LIN {X 0,Y 312.538,Z 248.086,A -85,B 0,C 180,E1 -15604.572,E2 -15604.572} C_VEL
LIN {X 0,Y 312.491,Z 248.051,A -85,B 0,C 180,E1 -15608.073,E2 -15608.073} C_VEL
LIN {X 0,Y 312.47,Z 248.049,A -85,B 0,C 180,E1 -15612.073,E2 -15612.073} C_VEL
LIN {X 0,Y 312.473,Z 248.051,A -85,B 0,C 180,E1 -15616.033,E2 -15616.033} C_VEL
LIN {X 0,Y 312.518,Z 248.056,A -85,B 0,C 180,E1 -15619.872,E2 -15619.872} C_VEL
LIN {X 0,Y 312.546,Z 248.05,A -85,B 0,C 180,E1 -15624.048,E2 -15624.048} C_VEL
LIN {X 0,Y 312.514,Z 248.051,A -85,B 0,C 180,E1 -15627.33,E2 -15627.33} C_VEL
LIN {X 0,Y 312.517,Z 248.049,A -85,B 0,C 180,E1 -15631.289,E2 -15631.289} C_VEL
LIN {X 0,Y 312.528,Z 248.053,A -85,B 0,C 180,E1 -15634.701,E2 -15634.701} C_VEL
LIN {X 0,Y 312.572,Z 248.052,A -85,B 0,C 180,E1 -15637.523,E2 -15637.523} C_VEL
LIN {X 0,Y 312.576,Z 248.049,A -85,B 0,C 180,E1 -15641.647,E2 -15641.647} C_VEL
LIN {X 0,Y 312.693,Z 248.029,A -85,B 0,C 180,E1 -15645.681,E2 -15645.681} C_VEL
LIN {X 0,Y 312.692,Z 248.025,A -85,B 0,C 180,E1 -15649.636,E2 -15649.636} C_VEL
LIN {X 0,Y 312.824,Z 248.015,A -85,B 0,C 180,E1 -15652.248,E2 -15652.248} C_VEL
LIN {X 0,Y 312.702,Z 248.028,A -85,B 0,C 180,E1 -15654.837,E2 -15654.837} C_VEL
LIN {X 0,Y 312.984,Z 247.987,A -85,B 0,C 180,E1 -15658.708,E2 -15658.708} C_VEL
LIN {X 0,Y 312.984,Z 247.997,A -85,B 0,C 180,E1 -15661.281,E2 -15661.281} C_VEL
LIN {X 0,Y 312.701,Z 248.033,A -85,B 0,C 180,E1 -15665.152,E2 -15665.152} C_VEL
LIN {X 0,Y 312.8,Z 248.01,A -85,B 0,C 180,E1 -15667.741,E2 -15667.741} C_VEL
LIN {X 0,Y 312.663,Z 248.028,A -85,B 0,C 180,E1 -15671.665,E2 -15671.665} C_VEL
LIN {X 0,Y 312.659,Z 248.032,A -85,B 0,C 180,E1 -15674.859,E2 -15674.859} C_VEL
LIN {X 0,Y 312.598,Z 248.042,A -85,B 0,C 180,E1 -15679.219,E2 -15679.219} C_VEL
LIN {X 0,Y 312.533,Z 248.052,A -85,B 0,C 180,E1 -15682.783,E2 -15682.783} C_VEL
LIN {X 0,Y 312.581,Z 248.026,A -85,B 0,C 180,E1 -15685.927,E2 -15685.927} C_VEL
LIN {X 0,Y 312.52,Z 248.052,A -85,B 0,C 180,E1 -15689.644,E2 -15689.644} C_VEL
LIN {X 0,Y 312.498,Z 248.057,A -85,B 0,C 180,E1 -15693.683,E2 -15693.683} C_VEL
LIN {X 0,Y 312.531,Z 248.05,A -85,B 0,C 180,E1 -15697.375,E2 -15697.375} C_VEL
LIN {X 0,Y 312.557,Z 248.173,A -85,B 0,C 180,E1 -15699.815,E2 -15699.815} C_VEL
LIN {X 0,Y 314.689,Z 256.545,A -85,B 0,C 180,E1 -15702.93,E2 -15702.93} C_VEL
LIN {X 0,Y 315.577,Z 260.265,A -85,B 0,C 180,E1 -15704.145,E2 -15704.145} C_VEL
LIN {X 0,Y 322.849,Z 275.668,A -85,B 0,C 180,E1 -15705.423,E2 -15705.423} C_VEL
LIN {X 0,Y 325.826,Z 282.967,A -85,B 0,C 180,E1 -15705.933,E2 -15705.933} C_VEL
LIN {X 0,Y 328.456,Z 295.565,A -85,B 0,C 180,E1 -15706.527,E2 -15706.527} C_VEL
LIN {X 0,Y 326.315,Z 367.557,A -85,B 0,C 180,E1 -15708.165,E2 -15708.165} C_VEL
LIN {X 0,Y 325.397,Z 380.734,A -85,B 0,C 180,E1 -15708.693,E2 -15708.693} C_VEL
LIN {X 0,Y 324.242,Z 393.12,A -85,B 0,C 180,E1 -15709.439,E2 -15709.439} C_VEL
LIN {X 0,Y 322.722,Z 405.254,A -85,B 0,C 180,E1 -15710.432,E2 -15710.432} C_VEL
LIN {X 0,Y 321.114,Z 416.236,A -85,B 0,C 180,E1 -15711.609,E2 -15711.609} C_VEL
LIN {X 0,Y 319.402,Z 426.332,A -85,B 0,C 180,E1 -15712.961,E2 -15712.961} C_VEL
LIN {X 0,Y 317.66,Z 435.593,A -85,B 0,C 180,E1 -15714.496,E2 -15714.496} C_VEL
LIN {X 0,Y 316.013,Z 443.977,A -85,B 0,C 180,E1 -15716.221,E2 -15716.221} C_VEL
LIN {X 0,Y 314.401,Z 451.459,A -85,B 0,C 180,E1 -15718.135,E2 -15718.135} C_VEL
LIN {X 0,Y 312.973,Z 458.38,A -85,B 0,C 180,E1 -15720.394,E2 -15720.394} C_VEL
LIN {X 0,Y 311.991,Z 463.287,A -85,B 0,C 180,E1 -15722.497,E2 -15722.497} C_VEL
LIN {X 0,Y 311.343,Z 466.913,A -85,B 0,C 180,E1 -15724.602,E2 -15724.602} C_VEL
LIN {X 0,Y 310.947,Z 468.671,A -85,B 0,C 180,E1 -15725.994,E2 -15725.994} C_VEL
LIN {X 0,Y 310.629,Z 470.416,A -85,B 0,C 180,E1 -15728.046,E2 -15728.046} C_VEL
LIN {X 0,Y 310.434,Z 471.174,A -85,B 0,C 180,E1 -15730.148,E2 -15730.148} C_VEL
LIN {X 0,Y 310.388,Z 471.006,A -85,B 0,C 180,E1 -15731.961,E2 -15731.961} C_VEL
LIN {X 0,Y 310.409,Z 469.679,A -85,B 0,C 180,E1 -15734.235,E2 -15734.235} C_VEL
LIN {X 0,Y 310.678,Z 467.044,A -85,B 0,C 180,E1 -15736.551,E2 -15736.551} C_VEL
LIN {X 0,Y 311.048,Z 462.897,A -85,B 0,C 180,E1 -15738.927,E2 -15738.927} C_VEL
LIN {X 0,Y 311.434,Z 458.154,A -85,B 0,C 180,E1 -15740.911,E2 -15740.911} C_VEL
LIN {X 0,Y 312.152,Z 451.86,A -85,B 0,C 180,E1 -15742.96,E2 -15742.96} C_VEL
LIN {X 0,Y 312.944,Z 444.608,A -85,B 0,C 180,E1 -15744.846,E2 -15744.846} C_VEL
LIN {X 0,Y 313.812,Z 436.952,A -85,B 0,C 180,E1 -15746.469,E2 -15746.469} C_VEL
LIN {X 0,Y 314.939,Z 427.65,A -85,B 0,C 180,E1 -15748.081,E2 -15748.081} C_VEL
LIN {X 0,Y 316.222,Z 416.808,A -85,B 0,C 180,E1 -15749.576,E2 -15749.576} C_VEL
LIN {X 0,Y 317.338,Z 405.733,A -85,B 0,C 180,E1 -15750.793,E2 -15750.793} C_VEL
LIN {X 0,Y 318.354,Z 393.728,A -85,B 0,C 180,E1 -15751.818,E2 -15751.818} C_VEL
LIN {X 0,Y 319.171,Z 381.15,A -85,B 0,C 180,E1 -15752.603,E2 -15752.603} C_VEL
LIN {X 0,Y 319.821,Z 368.153,A -85,B 0,C 180,E1 -15753.149,E2 -15753.149} C_VEL
LIN {X 0,Y 321.21,Z 306.929,A -85,B 0,C 180,E1 -15754.552,E2 -15754.552} C_VEL
LIN {X 0,Y 321.345,Z 291.631,A -85,B 0,C 180,E1 -15754.905,E2 -15754.905} C_VEL
LIN {X 0,Y 317.139,Z 266.964,A -85,B 0,C 180,E1 -15755.749,E2 -15755.749} C_VEL
LIN {X 0,Y 314.935,Z 260.111,A -85,B 0,C 180,E1 -15756.093,E2 -15756.093} C_VEL
LIN {X 0,Y 313.686,Z 252.533,A -85,B 0,C 180,E1 -15758.373,E2 -15758.373} C_VEL
LIN {X 0,Y 312.752,Z 248.06,A -85,B 0,C 180,E1 -15759.906,E2 -15759.906} C_VEL
LIN {X 0,Y 312.663,Z 248.034,A -85,B 0,C 180,E1 -15764.315,E2 -15764.315} C_VEL
LIN {X 0,Y 312.606,Z 248.027,A -85,B 0,C 180,E1 -15768.345,E2 -15768.345} C_VEL
LIN {X 0,Y 312.59,Z 248.047,A -85,B 0,C 180,E1 -15772.47,E2 -15772.47} C_VEL
LIN {X 0,Y 312.564,Z 248.018,A -85,B 0,C 180,E1 -15775.939,E2 -15775.939} C_VEL
LIN {X 0,Y 312.524,Z 248.044,A -85,B 0,C 180,E1 -15779.651,E2 -15779.651} C_VEL
LIN {X 0,Y 312.542,Z 248.048,A -85,B 0,C 180,E1 -15783.709,E2 -15783.709} C_VEL
LIN {X 0,Y 312.554,Z 248.049,A -85,B 0,C 180,E1 -15787.38,E2 -15787.38} C_VEL
LIN {X 0,Y 312.532,Z 248.048,A -85,B 0,C 180,E1 -15789.862,E2 -15789.862} C_VEL
LIN {X 0,Y 311.896,Z 248.126,A -85,B 0,C 180,E1 -15790.938,E2 -15790.938} C_VEL
LIN {X 0,Y 309.08,Z 248.479,A -85,B 0,C 180,E1 -15792.691,E2 -15792.691} C_VEL
LIN {X 0,Y 306.665,Z 248.781,A -85,B 0,C 180,E1 -15794.112,E2 -15794.112} C_VEL
LIN {X 0,Y 305.608,Z 248.913,A -85,B 0,C 180,E1 -15795.212,E2 -15795.212} C_VEL
LIN {X 0,Y 305.512,Z 248.925,A -85,B 0,C 180,E1 -15795.584,E2 -15795.584} C_VEL
LIN {X 0,Y 305.458,Z 248.925,A -85,B 0,C 180,E1 -15799.399,E2 -15799.399} C_VEL
LIN {X 0,Y 305.476,Z 248.918,A -85,B 0,C 180,E1 -15803.27,E2 -15803.27} C_VEL
LIN {X 0,Y 305.442,Z 248.939,A -85,B 0,C 180,E1 -15806.489,E2 -15806.489} C_VEL
LIN {X 0,Y 305.444,Z 248.926,A -85,B 0,C 180,E1 -15809.597,E2 -15809.597} C_VEL
LIN {X 0,Y 305.501,Z 248.895,A -85,B 0,C 180,E1 -15812.615,E2 -15812.615} C_VEL
LIN {X 0,Y 305.493,Z 248.922,A -85,B 0,C 180,E1 -15815.545,E2 -15815.545} C_VEL
LIN {X 0,Y 305.518,Z 248.923,A -85,B 0,C 180,E1 -15819.822,E2 -15819.822} C_VEL
LIN {X 0,Y 305.561,Z 248.899,A -85,B 0,C 180,E1 -15822.609,E2 -15822.609} C_VEL
LIN {X 0,Y 305.637,Z 248.874,A -85,B 0,C 180,E1 -15825.355,E2 -15825.355} C_VEL
LIN {X 0,Y 305.632,Z 248.91,A -85,B 0,C 180,E1 -15829.406,E2 -15829.406} C_VEL
LIN {X 0,Y 305.805,Z 248.889,A -85,B 0,C 180,E1 -15832.08,E2 -15832.08} C_VEL
LIN {X 0,Y 305.683,Z 248.895,A -85,B 0,C 180,E1 -15834.73,E2 -15834.73} C_VEL
LIN {X 0,Y 305.951,Z 248.838,A -85,B 0,C 180,E1 -15838.69,E2 -15838.69} C_VEL
LIN {X 0,Y 305.953,Z 248.861,A -85,B 0,C 180,E1 -15841.322,E2 -15841.322} C_VEL
LIN {X 0,Y 305.674,Z 248.907,A -85,B 0,C 180,E1 -15845.282,E2 -15845.282} C_VEL
LIN {X 0,Y 305.752,Z 248.88,A -85,B 0,C 180,E1 -15847.933,E2 -15847.933} C_VEL
LIN {X 0,Y 305.601,Z 248.893,A -85,B 0,C 180,E1 -15851.951,E2 -15851.951} C_VEL
LIN {X 0,Y 305.642,Z 248.91,A -85,B 0,C 180,E1 -15855.04,E2 -15855.04} C_VEL
LIN {X 0,Y 305.585,Z 248.906,A -85,B 0,C 180,E1 -15858.788,E2 -15858.788} C_VEL
LIN {X 0,Y 305.493,Z 248.921,A -85,B 0,C 180,E1 -15863.044,E2 -15863.044} C_VEL
LIN {X 0,Y 305.531,Z 248.928,A -85,B 0,C 180,E1 -15866.222,E2 -15866.222} C_VEL
LIN {X 0,Y 305.479,Z 248.915,A -85,B 0,C 180,E1 -15869.046,E2 -15869.046} C_VEL
LIN {X 0,Y 305.446,Z 248.933,A -85,B 0,C 180,E1 -15871.957,E2 -15871.957} C_VEL
LIN {X 0,Y 305.471,Z 248.933,A -85,B 0,C 180,E1 -15875.117,E2 -15875.117} C_VEL
LIN {X 0,Y 305.445,Z 248.93,A -85,B 0,C 180,E1 -15878.529,E2 -15878.529} C_VEL
LIN {X 0,Y 305.451,Z 248.928,A -85,B 0,C 180,E1 -15881.861,E2 -15881.861} C_VEL
LIN {X 0,Y 305.411,Z 248.902,A -85,B 0,C 180,E1 -15885.515,E2 -15885.515} C_VEL
LIN {X 0,Y 305.424,Z 248.934,A -85,B 0,C 180,E1 -15888.141,E2 -15888.141} C_VEL
LIN {X 0,Y 305.457,Z 248.925,A -85,B 0,C 180,E1 -15891.595,E2 -15891.595} C_VEL
LIN {X 0,Y 305.475,Z 248.932,A -85,B 0,C 180,E1 -15894.889,E2 -15894.889} C_VEL
LIN {X 0,Y 305.456,Z 248.932,A -85,B 0,C 180,E1 -15898.361,E2 -15898.361} C_VEL
LIN {X 0,Y 305.56,Z 249.121,A -85,B 0,C 180,E1 -15899.775,E2 -15899.775} C_VEL
LIN {X 0,Y 307.636,Z 259.297,A -85,B 0,C 180,E1 -15903.002,E2 -15903.002} C_VEL
LIN {X 0,Y 308.973,Z 267.763,A -85,B 0,C 180,E1 -15905.519,E2 -15905.519} C_VEL
LIN {X 0,Y 309.608,Z 272.24,A -85,B 0,C 180,E1 -15905.741,E2 -15905.741} C_VEL
LIN {X 0,Y 314.56,Z 305.462,A -85,B 0,C 180,E1 -15906.861,E2 -15906.861} C_VEL
LIN {X 0,Y 313.094,Z 375.459,A -85,B 0,C 180,E1 -15908.478,E2 -15908.478} C_VEL
LIN {X 0,Y 312.383,Z 388.794,A -85,B 0,C 180,E1 -15909.032,E2 -15909.032} C_VEL
LIN {X 0,Y 311.352,Z 402.15,A -85,B 0,C 180,E1 -15909.866,E2 -15909.866} C_VEL
LIN {X 0,Y 310.293,Z 413.361,A -85,B 0,C 180,E1 -15910.828,E2 -15910.828} C_VEL
LIN {X 0,Y 308.976,Z 425.009,A -85,B 0,C 180,E1 -15912.118,E2 -15912.118} C_VEL
LIN {X 0,Y 307.955,Z 434.567,A -85,B 0,C 180,E1 -15913.448,E2 -15913.448} C_VEL
LIN {X 0,Y 306.817,Z 444.067,A -85,B 0,C 180,E1 -15915.067,E2 -15915.067} C_VEL
LIN {X 0,Y 305.827,Z 451.94,A -85,B 0,C 180,E1 -15916.715,E2 -15916.715} C_VEL
LIN {X 0,Y 304.915,Z 459.611,A -85,B 0,C 180,E1 -15918.702,E2 -15918.702} C_VEL
LIN {X 0,Y 304.275,Z 465.769,A -85,B 0,C 180,E1 -15920.696,E2 -15920.696} C_VEL
LIN {X 0,Y 303.857,Z 470.636,A -85,B 0,C 180,E1 -15922.692,E2 -15922.692} C_VEL
LIN {X 0,Y 303.634,Z 474.361,A -85,B 0,C 180,E1 -15924.688,E2 -15924.688} C_VEL
LIN {X 0,Y 303.594,Z 476.281,A -85,B 0,C 180,E1 -15926.018,E2 -15926.018} C_VEL
LIN {X 0,Y 303.588,Z 477.755,A -85,B 0,C 180,E1 -15927.347,E2 -15927.347} C_VEL
LIN {X 0,Y 303.537,Z 478.786,A -85,B 0,C 180,E1 -15928.674,E2 -15928.674} C_VEL
LIN {X 0,Y 303.543,Z 479.428,A -85,B 0,C 180,E1 -15930,E2 -15930} C_VEL
LIN {X 0,Y 303.536,Z 479.683,A -85,B 0,C 180,E1 -15931.327,E2 -15931.327} C_VEL
LIN {X 0,Y 303.591,Z 479.534,A -85,B 0,C 180,E1 -15932.654,E2 -15932.654} C_VEL
LIN {X 0,Y 303.703,Z 478.009,A -85,B 0,C 180,E1 -15935.312,E2 -15935.312} C_VEL
LIN {X 0,Y 303.855,Z 476.667,A -85,B 0,C 180,E1 -15936.641,E2 -15936.641} C_VEL
LIN {X 0,Y 304.308,Z 473.841,A -85,B 0,C 180,E1 -15938.634,E2 -15938.634} C_VEL
LIN {X 0,Y 305.043,Z 470.011,A -85,B 0,C 180,E1 -15940.622,E2 -15940.622} C_VEL
LIN {X 0,Y 306.06,Z 465.078,A -85,B 0,C 180,E1 -15942.601,E2 -15942.601} C_VEL
LIN {X 0,Y 307.378,Z 458.897,A -85,B 0,C 180,E1 -15944.567,E2 -15944.567} C_VEL
LIN {X 0,Y 309.075,Z 451.207,A -85,B 0,C 180,E1 -15946.514,E2 -15946.514} C_VEL
LIN {X 0,Y 310.657,Z 442.8,A -85,B 0,C 180,E1 -15948.236,E2 -15948.236} C_VEL
LIN {X 0,Y 312.614,Z 432.788,A -85,B 0,C 180,E1 -15949.879,E2 -15949.879} C_VEL
LIN {X 0,Y 314.599,Z 421.985,A -85,B 0,C 180,E1 -15951.286,E2 -15951.286} C_VEL
LIN {X 0,Y 316.245,Z 411.445,A -85,B 0,C 180,E1 -15952.37,E2 -15952.37} C_VEL
LIN {X 0,Y 317.928,Z 398.798,A -85,B 0,C 180,E1 -15953.361,E2 -15953.361} C_VEL
LIN {X 0,Y 319.224,Z 386.15,A -85,B 0,C 180,E1 -15954.078,E2 -15954.078} C_VEL
LIN {X 0,Y 320.088,Z 372.579,A -85,B 0,C 180,E1 -15954.57,E2 -15954.57} C_VEL
LIN {X 0,Y 321.971,Z 308.158,A -85,B 0,C 180,E1 -15956.059,E2 -15956.059} C_VEL
LIN {X 0,Y 318.94,Z 292.083,A -85,B 0,C 180,E1 -15956.812,E2 -15956.812} C_VEL
LIN {X 0,Y 316.695,Z 282.309,A -85,B 0,C 180,E1 -15957.325,E2 -15957.325} C_VEL
LIN {X 0,Y 310.968,Z 269.796,A -85,B 0,C 180,E1 -15958.344,E2 -15958.344} C_VEL
LIN {X 0,Y 309.964,Z 267.204,A -85,B 0,C 180,E1 -15958.619,E2 -15958.619} C_VEL
LIN {X 0,Y 307.884,Z 258.403,A -85,B 0,C 180,E1 -15961.67,E2 -15961.67} C_VEL
LIN {X 0,Y 305.531,Z 249.134,A -85,B 0,C 180,E1 -15965.205,E2 -15965.205} C_VEL
LIN {X 0,Y 305.449,Z 248.925,A -85,B 0,C 180,E1 -15968.523,E2 -15968.523} C_VEL
LIN {X 0,Y 305.45,Z 248.921,A -85,B 0,C 180,E1 -15972.579,E2 -15972.579} C_VEL
LIN {X 0,Y 305.438,Z 248.922,A -85,B 0,C 180,E1 -15976.341,E2 -15976.341} C_VEL
LIN {X 0,Y 305.472,Z 248.934,A -85,B 0,C 180,E1 -15979.889,E2 -15979.889} C_VEL
LIN {X 0,Y 305.476,Z 248.932,A -85,B 0,C 180,E1 -15983.633,E2 -15983.633} C_VEL
LIN {X 0,Y 305.478,Z 248.935,A -85,B 0,C 180,E1 -15986.48,E2 -15986.48} C_VEL
LIN {X 0,Y 305.442,Z 248.938,A -85,B 0,C 180,E1 -15989.583,E2 -15989.583} C_VEL
LIN {X 0,Y 305.462,Z 248.929,A -85,B 0,C 180,E1 -15992.598,E2 -15992.598} C_VEL
LIN {X 0,Y 305.451,Z 248.927,A -85,B 0,C 180,E1 -15995.529,E2 -15995.529} C_VEL
LIN {X 0,Y 305.493,Z 248.921,A -85,B 0,C 180,E1 -15999.808,E2 -15999.808} C_VEL
LIN {X 0,Y 305.559,Z 248.912,A -85,B 0,C 180,E1 -16003.973,E2 -16003.973} C_VEL
LIN {X 0,Y 305.594,Z 248.917,A -85,B 0,C 180,E1 -16006.699,E2 -16006.699} C_VEL
LIN {X 0,Y 305.758,Z 248.897,A -85,B 0,C 180,E1 -16011.256,E2 -16011.256} C_VEL
LIN {X 0,Y 305.803,Z 248.884,A -85,B 0,C 180,E1 -16013.396,E2 -16013.396} C_VEL
LIN {X 0,Y 305.951,Z 248.863,A -85,B 0,C 180,E1 -16018.678,E2 -16018.678} C_VEL
LIN {X 0,Y 305.951,Z 248.874,A -85,B 0,C 180,E1 -16021.31,E2 -16021.31} C_VEL
LIN {X 0,Y 305.67,Z 248.908,A -85,B 0,C 180,E1 -16025.271,E2 -16025.271} C_VEL
LIN {X 0,Y 305.749,Z 248.89,A -85,B 0,C 180,E1 -16027.921,E2 -16027.921} C_VEL
LIN {X 0,Y 305.597,Z 248.909,A -85,B 0,C 180,E1 -16031.939,E2 -16031.939} C_VEL
LIN {X 0,Y 305.601,Z 248.91,A -85,B 0,C 180,E1 -16035.008,E2 -16035.008} C_VEL
LIN {X 0,Y 305.55,Z 248.921,A -85,B 0,C 180,E1 -16039.43,E2 -16039.43} C_VEL
LIN {X 0,Y 305.477,Z 248.933,A -85,B 0,C 180,E1 -16043.035,E2 -16043.035} C_VEL
LIN {X 0,Y 305.51,Z 248.906,A -85,B 0,C 180,E1 -16046.212,E2 -16046.212} C_VEL
LIN {X 0,Y 305.471,Z 248.935,A -85,B 0,C 180,E1 -16049.041,E2 -16049.041} C_VEL
LIN {X 0,Y 305.422,Z 248.929,A -85,B 0,C 180,E1 -16051.946,E2 -16051.946} C_VEL
LIN {X 0,Y 305.441,Z 248.926,A -85,B 0,C 180,E1 -16055.107,E2 -16055.107} C_VEL
LIN {X 0,Y 305.493,Z 249.04,A -85,B 0,C 180,E1 -16059.044,E2 -16059.044} C_VEL
LIN {X 0,Y 307.721,Z 257.568,A -85,B 0,C 180,E1 -16062.347,E2 -16062.347} C_VEL
LIN {X 0,Y 308.401,Z 260.473,A -85,B 0,C 180,E1 -16063.287,E2 -16063.287} C_VEL
LIN {X 0,Y 315.715,Z 275.48,A -85,B 0,C 180,E1 -16064.615,E2 -16064.615} C_VEL
LIN {X 0,Y 320.159,Z 285.993,A -85,B 0,C 180,E1 -16065.398,E2 -16065.398} C_VEL
LIN {X 0,Y 322.355,Z 296.98,A -85,B 0,C 180,E1 -16065.926,E2 -16065.926} C_VEL
LIN {X 0,Y 320.052,Z 368.301,A -85,B 0,C 180,E1 -16067.58,E2 -16067.58} C_VEL
LIN {X 0,Y 319.119,Z 381.269,A -85,B 0,C 180,E1 -16068.119,E2 -16068.119} C_VEL
LIN {X 0,Y 317.901,Z 393.543,A -85,B 0,C 180,E1 -16068.876,E2 -16068.876} C_VEL
LIN {X 0,Y 316.317,Z 405.571,A -85,B 0,C 180,E1 -16069.884,E2 -16069.884} C_VEL
LIN {X 0,Y 314.642,Z 416.512,A -85,B 0,C 180,E1 -16071.081,E2 -16071.081} C_VEL
LIN {X 0,Y 312.811,Z 426.726,A -85,B 0,C 180,E1 -16072.479,E2 -16072.479} C_VEL
LIN {X 0,Y 311.017,Z 435.806,A -85,B 0,C 180,E1 -16074.019,E2 -16074.019} C_VEL
LIN {X 0,Y 309.284,Z 444.162,A -85,B 0,C 180,E1 -16075.777,E2 -16075.777} C_VEL
LIN {X 0,Y 307.631,Z 451.479,A -85,B 0,C 180,E1 -16077.687,E2 -16077.687} C_VEL
LIN {X 0,Y 306.28,Z 457.565,A -85,B 0,C 180,E1 -16079.68,E2 -16079.68} C_VEL
LIN {X 0,Y 305.192,Z 462.685,A -85,B 0,C 180,E1 -16081.831,E2 -16081.831} C_VEL
LIN {X 0,Y 304.345,Z 466.871,A -85,B 0,C 180,E1 -16084.217,E2 -16084.217} C_VEL
LIN {X 0,Y 303.711,Z 469.799,A -85,B 0,C 180,E1 -16086.834,E2 -16086.834} C_VEL
LIN {X 0,Y 303.519,Z 470.755,A -85,B 0,C 180,E1 -16088.254,E2 -16088.254} C_VEL
LIN {X 0,Y 303.356,Z 471.235,A -85,B 0,C 180,E1 -16089.664,E2 -16089.664} C_VEL
LIN {X 0,Y 303.286,Z 471.129,A -85,B 0,C 180,E1 -16091.794,E2 -16091.794} C_VEL
LIN {X 0,Y 303.286,Z 470.06,A -85,B 0,C 180,E1 -16093.854,E2 -16093.854} C_VEL
LIN {X 0,Y 303.558,Z 467.261,A -85,B 0,C 180,E1 -16096.467,E2 -16096.467} C_VEL
LIN {X 0,Y 303.901,Z 463.626,A -85,B 0,C 180,E1 -16098.663,E2 -16098.663} C_VEL
LIN {X 0,Y 304.272,Z 459.084,A -85,B 0,C 180,E1 -16100.695,E2 -16100.695} C_VEL
LIN {X 0,Y 305.032,Z 452.698,A -85,B 0,C 180,E1 -16102.895,E2 -16102.895} C_VEL
LIN {X 0,Y 305.949,Z 444.637,A -85,B 0,C 180,E1 -16105.058,E2 -16105.058} C_VEL
LIN {X 0,Y 306.85,Z 436.967,A -85,B 0,C 180,E1 -16106.717,E2 -16106.717} C_VEL
LIN {X 0,Y 307.994,Z 427.65,A -85,B 0,C 180,E1 -16108.365,E2 -16108.365} C_VEL
LIN {X 0,Y 309.308,Z 417.08,A -85,B 0,C 180,E1 -16109.853,E2 -16109.853} C_VEL
LIN {X 0,Y 310.48,Z 405.663,A -85,B 0,C 180,E1 -16111.134,E2 -16111.134} C_VEL
LIN {X 0,Y 311.54,Z 393.581,A -85,B 0,C 180,E1 -16112.181,E2 -16112.181} C_VEL
LIN {X 0,Y 312.386,Z 380.901,A -85,B 0,C 180,E1 -16112.982,E2 -16112.982} C_VEL
LIN {X 0,Y 313.068,Z 367.718,A -85,B 0,C 180,E1 -16113.539,E2 -16113.539} C_VEL
LIN {X 0,Y 314.735,Z 293.135,A -85,B 0,C 180,E1 -16115.27,E2 -16115.27} C_VEL
LIN {X 0,Y 310.542,Z 268.816,A -85,B 0,C 180,E1 -16116.124,E2 -16116.124} C_VEL
LIN {X 0,Y 307.846,Z 260.311,A -85,B 0,C 180,E1 -16116.554,E2 -16116.554} C_VEL
LIN {X 0,Y 307.24,Z 256.803,A -85,B 0,C 180,E1 -16117.557,E2 -16117.557} C_VEL
LIN {X 0,Y 305.723,Z 248.994,A -85,B 0,C 180,E1 -16120.178,E2 -16120.178} C_VEL
LIN {X 0,Y 305.606,Z 248.913,A -85,B 0,C 180,E1 -16125.045,E2 -16125.045} C_VEL
LIN {X 0,Y 305.572,Z 248.898,A -85,B 0,C 180,E1 -16129.467,E2 -16129.467} C_VEL
LIN {X 0,Y 305.514,Z 248.929,A -85,B 0,C 180,E1 -16133.073,E2 -16133.073} C_VEL
LIN {X 0,Y 305.509,Z 248.893,A -85,B 0,C 180,E1 -16136.231,E2 -16136.231} C_VEL
LIN {X 0,Y 305.474,Z 248.914,A -85,B 0,C 180,E1 -16139.06,E2 -16139.06} C_VEL
LIN {X 0,Y 305.466,Z 248.937,A -85,B 0,C 180,E1 -16141.949,E2 -16141.949} C_VEL
LIN {X 0,Y 305.494,Z 248.919,A -85,B 0,C 180,E1 -16145.108,E2 -16145.108} C_VEL
LIN {X 0,Y 305.506,Z 248.928,A -85,B 0,C 180,E1 -16148.555,E2 -16148.555} C_VEL
LIN {X 0,Y 305.504,Z 248.909,A -85,B 0,C 180,E1 -16152.607,E2 -16152.607} C_VEL
LIN {X 0,Y 305.512,Z 248.925,A -85,B 0,C 180,E1 -16155.584,E2 -16155.584} C_VEL
LIN {X 0,Y 304.814,Z 249.015,A -85,B 0,C 180,E1 -16156.684,E2 -16156.684} C_VEL
LIN {X 0,Y 301.938,Z 249.366,A -85,B 0,C 180,E1 -16158.473,E2 -16158.473} C_VEL
LIN {X 0,Y 299.517,Z 249.655,A -85,B 0,C 180,E1 -16159.925,E2 -16159.925} C_VEL
LIN {X 0,Y 298.481,Z 249.776,A -85,B 0,C 180,E1 -16161.049,E2 -16161.049} C_VEL
LIN {X 0,Y 298.397,Z 249.785,A -85,B 0,C 180,E1 -16161.43,E2 -16161.43} C_VEL
LIN {X 0,Y 298.408,Z 249.802,A -85,B 0,C 180,E1 -16163.938,E2 -16163.938} C_VEL
LIN {X 0,Y 298.376,Z 249.817,A -85,B 0,C 180,E1 -16167.988,E2 -16167.988} C_VEL
LIN {X 0,Y 298.443,Z 249.774,A -85,B 0,C 180,E1 -16171.911,E2 -16171.911} C_VEL
LIN {X 0,Y 298.469,Z 249.79,A -85,B 0,C 180,E1 -16174.93,E2 -16174.93} C_VEL
LIN {X 0,Y 298.452,Z 249.805,A -85,B 0,C 180,E1 -16179.323,E2 -16179.323} C_VEL
LIN {X 0,Y 298.525,Z 249.782,A -85,B 0,C 180,E1 -16182.186,E2 -16182.186} C_VEL
LIN {X 0,Y 298.581,Z 249.751,A -85,B 0,C 180,E1 -16185.001,E2 -16185.001} C_VEL
LIN {X 0,Y 298.586,Z 249.784,A -85,B 0,C 180,E1 -16189.153,E2 -16189.153} C_VEL
LIN {X 0,Y 298.751,Z 249.768,A -85,B 0,C 180,E1 -16191.892,E2 -16191.892} C_VEL
LIN {X 0,Y 298.654,Z 249.77,A -85,B 0,C 180,E1 -16194.605,E2 -16194.605} C_VEL
LIN {X 0,Y 298.918,Z 249.713,A -85,B 0,C 180,E1 -16198.659,E2 -16198.659} C_VEL
LIN {X 0,Y 298.919,Z 249.737,A -85,B 0,C 180,E1 -16201.353,E2 -16201.353} C_VEL
LIN {X 0,Y 298.642,Z 249.784,A -85,B 0,C 180,E1 -16205.407,E2 -16205.407} C_VEL
LIN {X 0,Y 298.703,Z 249.755,A -85,B 0,C 180,E1 -16208.121,E2 -16208.121} C_VEL
LIN {X 0,Y 298.553,Z 249.774,A -85,B 0,C 180,E1 -16212.237,E2 -16212.237} C_VEL
LIN {X 0,Y 298.61,Z 249.786,A -85,B 0,C 180,E1 -16215.214,E2 -16215.214} C_VEL
LIN {X 0,Y 298.531,Z 249.782,A -85,B 0,C 180,E1 -16219.249,E2 -16219.249} C_VEL
LIN {X 0,Y 298.436,Z 249.804,A -85,B 0,C 180,E1 -16223.605,E2 -16223.605} C_VEL
LIN {X 0,Y 298.491,Z 249.806,A -85,B 0,C 180,E1 -16226.58,E2 -16226.58} C_VEL
LIN {X 0,Y 298.412,Z 249.792,A -85,B 0,C 180,E1 -16229.647,E2 -16229.647} C_VEL
LIN {X 0,Y 298.402,Z 249.815,A -85,B 0,C 180,E1 -16232.805,E2 -16232.805} C_VEL
LIN {X 0,Y 298.438,Z 249.799,A -85,B 0,C 180,E1 -16236.806,E2 -16236.806} C_VEL
LIN {X 0,Y 298.398,Z 249.815,A -85,B 0,C 180,E1 -16241.091,E2 -16241.091} C_VEL
LIN {X 0,Y 298.411,Z 249.79,A -85,B 0,C 180,E1 -16243.107,E2 -16243.107} C_VEL
LIN {X 0,Y 298.383,Z 249.794,A -85,B 0,C 180,E1 -16246.918,E2 -16246.918} C_VEL
LIN {X 0,Y 298.366,Z 249.812,A -85,B 0,C 180,E1 -16251.022,E2 -16251.022} C_VEL
LIN {X 0,Y 298.418,Z 249.815,A -85,B 0,C 180,E1 -16253.931,E2 -16253.931} C_VEL
LIN {X 0,Y 298.407,Z 249.815,A -85,B 0,C 180,E1 -16257.202,E2 -16257.202} C_VEL
LIN {X 0,Y 298.47,Z 249.919,A -85,B 0,C 180,E1 -16259.391,E2 -16259.391} C_VEL
LIN {X 0,Y 300.562,Z 260.037,A -85,B 0,C 180,E1 -16262.699,E2 -16262.699} C_VEL
LIN {X 0,Y 301.934,Z 267.798,A -85,B 0,C 180,E1 -16265.057,E2 -16265.057} C_VEL
LIN {X 0,Y 302.81,Z 272.446,A -85,B 0,C 180,E1 -16265.286,E2 -16265.286} C_VEL
LIN {X 0,Y 307.872,Z 307.326,A -85,B 0,C 180,E1 -16266.489,E2 -16266.489} C_VEL
LIN {X 0,Y 306.296,Z 375.768,A -85,B 0,C 180,E1 -16268.109,E2 -16268.109} C_VEL
LIN {X 0,Y 305.553,Z 388.961,A -85,B 0,C 180,E1 -16268.673,E2 -16268.673} C_VEL
LIN {X 0,Y 304.54,Z 401.688,A -85,B 0,C 180,E1 -16269.483,E2 -16269.483} C_VEL
LIN {X 0,Y 303.368,Z 413.801,A -85,B 0,C 180,E1 -16270.548,E2 -16270.548} C_VEL
LIN {X 0,Y 302.017,Z 425.355,A -85,B 0,C 180,E1 -16271.867,E2 -16271.867} C_VEL
LIN {X 0,Y 300.968,Z 434.854,A -85,B 0,C 180,E1 -16273.229,E2 -16273.229} C_VEL
LIN {X 0,Y 299.939,Z 443.389,A -85,B 0,C 180,E1 -16274.717,E2 -16274.717} C_VEL
LIN {X 0,Y 298.89,Z 451.373,A -85,B 0,C 180,E1 -16276.401,E2 -16276.401} C_VEL
LIN {X 0,Y 297.901,Z 459.151,A -85,B 0,C 180,E1 -16278.433,E2 -16278.433} C_VEL
LIN {X 0,Y 297.245,Z 465.381,A -85,B 0,C 180,E1 -16280.474,E2 -16280.474} C_VEL
LIN {X 0,Y 296.805,Z 470.312,A -85,B 0,C 180,E1 -16282.517,E2 -16282.517} C_VEL
LIN {X 0,Y 296.549,Z 474.094,A -85,B 0,C 180,E1 -16284.561,E2 -16284.561} C_VEL
LIN {X 0,Y 296.496,Z 476.041,A -85,B 0,C 180,E1 -16285.923,E2 -16285.923} C_VEL
LIN {X 0,Y 296.493,Z 477.562,A -85,B 0,C 180,E1 -16287.283,E2 -16287.283} C_VEL
LIN {X 0,Y 296.458,Z 478.625,A -85,B 0,C 180,E1 -16288.642,E2 -16288.642} C_VEL
LIN {X 0,Y 296.462,Z 479.291,A -85,B 0,C 180,E1 -16290,E2 -16290} C_VEL
LIN {X 0,Y 296.458,Z 479.571,A -85,B 0,C 180,E1 -16291.359,E2 -16291.359} C_VEL
LIN {X 0,Y 296.496,Z 479.464,A -85,B 0,C 180,E1 -16292.718,E2 -16292.718} C_VEL
LIN {X 0,Y 296.618,Z 478.002,A -85,B 0,C 180,E1 -16295.439,E2 -16295.439} C_VEL
LIN {X 0,Y 297.079,Z 474.971,A -85,B 0,C 180,E1 -16298.161,E2 -16298.161} C_VEL
LIN {X 0,Y 297.785,Z 471.539,A -85,B 0,C 180,E1 -16300.196,E2 -16300.196} C_VEL
LIN {X 0,Y 298.747,Z 467.049,A -85,B 0,C 180,E1 -16302.224,E2 -16302.224} C_VEL
LIN {X 0,Y 300.221,Z 460.274,A -85,B 0,C 180,E1 -16304.576,E2 -16304.576} C_VEL
LIN {X 0,Y 301.988,Z 452.932,A -85,B 0,C 180,E1 -16306.564,E2 -16306.564} C_VEL
LIN {X 0,Y 303.627,Z 444.778,A -85,B 0,C 180,E1 -16308.363,E2 -16308.363} C_VEL
LIN {X 0,Y 305.557,Z 435.504,A -85,B 0,C 180,E1 -16310.007,E2 -16310.007} C_VEL
LIN {X 0,Y 307.605,Z 425.314,A -85,B 0,C 180,E1 -16311.442,E2 -16311.442} C_VEL
LIN {X 0,Y 309.501,Z 414.063,A -85,B 0,C 180,E1 -16312.708,E2 -16312.708} C_VEL
LIN {X 0,Y 311.271,Z 402.382,A -85,B 0,C 180,E1 -16313.715,E2 -16313.715} C_VEL
LIN {X 0,Y 312.598,Z 390.375,A -85,B 0,C 180,E1 -16314.49,E2 -16314.49} C_VEL
LIN {X 0,Y 313.678,Z 377.213,A -85,B 0,C 180,E1 -16315.062,E2 -16315.062} C_VEL
LIN {X 0,Y 314.538,Z 352.517,A -85,B 0,C 180,E1 -16315.688,E2 -16315.688} C_VEL
LIN {X 0,Y 315.884,Z 309.406,A -85,B 0,C 180,E1 -16316.69,E2 -16316.69} C_VEL
LIN {X 0,Y 313.161,Z 294.664,A -85,B 0,C 180,E1 -16317.397,E2 -16317.397} C_VEL
LIN {X 0,Y 311.121,Z 285.489,A -85,B 0,C 180,E1 -16317.888,E2 -16317.888} C_VEL
LIN {X 0,Y 304.482,Z 270.92,A -85,B 0,C 180,E1 -16319.12,E2 -16319.12} C_VEL
LIN {X 0,Y 302.736,Z 267.207,A -85,B 0,C 180,E1 -16319.513,E2 -16319.513} C_VEL
LIN {X 0,Y 300.631,Z 258.379,A -85,B 0,C 180,E1 -16322.685,E2 -16322.685} C_VEL
LIN {X 0,Y 298.483,Z 249.933,A -85,B 0,C 180,E1 -16326.061,E2 -16326.061} C_VEL
LIN {X 0,Y 298.39,Z 249.807,A -85,B 0,C 180,E1 -16329.49,E2 -16329.49} C_VEL
LIN {X 0,Y 298.385,Z 249.802,A -85,B 0,C 180,E1 -16333.094,E2 -16333.094} C_VEL
LIN {X 0,Y 298.39,Z 249.795,A -85,B 0,C 180,E1 -16336.913,E2 -16336.913} C_VEL
LIN {X 0,Y 298.404,Z 249.81,A -85,B 0,C 180,E1 -16341.007,E2 -16341.007} C_VEL
LIN {X 0,Y 298.418,Z 249.811,A -85,B 0,C 180,E1 -16343.925,E2 -16343.925} C_VEL
LIN {X 0,Y 298.406,Z 249.81,A -85,B 0,C 180,E1 -16347.196,E2 -16347.196} C_VEL
LIN {X 0,Y 298.413,Z 249.812,A -85,B 0,C 180,E1 -16350.622,E2 -16350.622} C_VEL
LIN {X 0,Y 298.425,Z 249.806,A -85,B 0,C 180,E1 -16354.913,E2 -16354.913} C_VEL
LIN {X 0,Y 298.409,Z 249.814,A -85,B 0,C 180,E1 -16357.857,E2 -16357.857} C_VEL
LIN {X 0,Y 298.474,Z 249.796,A -85,B 0,C 180,E1 -16360.747,E2 -16360.747} C_VEL
LIN {X 0,Y 298.594,Z 249.778,A -85,B 0,C 180,E1 -16364.989,E2 -16364.989} C_VEL
LIN {X 0,Y 298.59,Z 249.78,A -85,B 0,C 180,E1 -16369.141,E2 -16369.141} C_VEL
LIN {X 0,Y 298.715,Z 249.776,A -85,B 0,C 180,E1 -16371.879,E2 -16371.879} C_VEL
LIN {X 0,Y 298.641,Z 249.777,A -85,B 0,C 180,E1 -16374.593,E2 -16374.593} C_VEL
LIN {X 0,Y 298.917,Z 249.739,A -85,B 0,C 180,E1 -16378.647,E2 -16378.647} C_VEL
LIN {X 0,Y 298.918,Z 249.75,A -85,B 0,C 180,E1 -16381.341,E2 -16381.341} C_VEL
LIN {X 0,Y 298.71,Z 249.767,A -85,B 0,C 180,E1 -16386.507,E2 -16386.507} C_VEL
LIN {X 0,Y 298.626,Z 249.786,A -85,B 0,C 180,E1 -16389.476,E2 -16389.476} C_VEL
LIN {X 0,Y 298.538,Z 249.797,A -85,B 0,C 180,E1 -16393.609,E2 -16393.609} C_VEL
LIN {X 0,Y 298.478,Z 249.802,A -85,B 0,C 180,E1 -16396.406,E2 -16396.406} C_VEL
LIN {X 0,Y 298.488,Z 249.802,A -85,B 0,C 180,E1 -16399.641,E2 -16399.641} C_VEL
LIN {X 0,Y 298.444,Z 249.81,A -85,B 0,C 180,E1 -16403.591,E2 -16403.591} C_VEL
LIN {X 0,Y 298.468,Z 249.783,A -85,B 0,C 180,E1 -16406.568,E2 -16406.568} C_VEL
LIN {X 0,Y 298.398,Z 249.81,A -85,B 0,C 180,E1 -16409.635,E2 -16409.635} C_VEL
LIN {X 0,Y 298.374,Z 249.818,A -85,B 0,C 180,E1 -16412.794,E2 -16412.794} C_VEL
LIN {X 0,Y 298.448,Z 249.812,A -85,B 0,C 180,E1 -16416.808,E2 -16416.808} C_VEL
LIN {X 0,Y 298.471,Z 249.985,A -85,B 0,C 180,E1 -16418.287,E2 -16418.287} C_VEL
LIN {X 0,Y 300.952,Z 259.501,A -85,B 0,C 180,E1 -16422.063,E2 -16422.063} C_VEL
LIN {X 0,Y 301.392,Z 260.902,A -85,B 0,C 180,E1 -16422.401,E2 -16422.401} C_VEL
LIN {X 0,Y 309.22,Z 276.687,A -85,B 0,C 180,E1 -16423.874,E2 -16423.874} C_VEL
LIN {X 0,Y 314.369,Z 288.532,A -85,B 0,C 180,E1 -16424.811,E2 -16424.811} C_VEL
LIN {X 0,Y 316.275,Z 297.985,A -85,B 0,C 180,E1 -16425.283,E2 -16425.283} C_VEL
LIN {X 0,Y 313.917,Z 368.086,A -85,B 0,C 180,E1 -16426.934,E2 -16426.934} C_VEL
LIN {X 0,Y 312.934,Z 381.128,A -85,B 0,C 180,E1 -16427.479,E2 -16427.479} C_VEL
LIN {X 0,Y 311.611,Z 393.944,A -85,B 0,C 180,E1 -16428.282,E2 -16428.282} C_VEL
LIN {X 0,Y 309.953,Z 405.946,A -85,B 0,C 180,E1 -16429.316,E2 -16429.316} C_VEL
LIN {X 0,Y 308.183,Z 416.947,A -85,B 0,C 180,E1 -16430.548,E2 -16430.548} C_VEL
LIN {X 0,Y 306.306,Z 426.823,A -85,B 0,C 180,E1 -16431.929,E2 -16431.929} C_VEL
LIN {X 0,Y 304.505,Z 435.472,A -85,B 0,C 180,E1 -16433.419,E2 -16433.419} C_VEL
LIN {X 0,Y 302.591,Z 444.351,A -85,B 0,C 180,E1 -16435.316,E2 -16435.316} C_VEL
LIN {X 0,Y 300.665,Z 452.358,A -85,B 0,C 180,E1 -16437.478,E2 -16437.478} C_VEL
LIN {X 0,Y 299.206,Z 458.695,A -85,B 0,C 180,E1 -16439.668,E2 -16439.668} C_VEL
LIN {X 0,Y 298.073,Z 463.562,A -85,B 0,C 180,E1 -16441.864,E2 -16441.864} C_VEL
LIN {X 0,Y 297.363,Z 466.933,A -85,B 0,C 180,E1 -16443.891,E2 -16443.891} C_VEL
LIN {X 0,Y 296.723,Z 469.621,A -85,B 0,C 180,E1 -16446.256,E2 -16446.256} C_VEL
LIN {X 0,Y 296.498,Z 470.659,A -85,B 0,C 180,E1 -16447.712,E2 -16447.712} C_VEL
LIN {X 0,Y 296.3,Z 471.268,A -85,B 0,C 180,E1 -16449.158,E2 -16449.158} C_VEL
LIN {X 0,Y 296.208,Z 471.254,A -85,B 0,C 180,E1 -16451.606,E2 -16451.606} C_VEL
LIN {X 0,Y 296.182,Z 470.384,A -85,B 0,C 180,E1 -16453.456,E2 -16453.456} C_VEL
LIN {X 0,Y 296.268,Z 469.227,A -85,B 0,C 180,E1 -16454.874,E2 -16454.874} C_VEL
LIN {X 0,Y 296.443,Z 467.476,A -85,B 0,C 180,E1 -16456.377,E2 -16456.377} C_VEL
LIN {X 0,Y 296.779,Z 464.321,A -85,B 0,C 180,E1 -16458.387,E2 -16458.387} C_VEL
LIN {X 0,Y 297.145,Z 459.952,A -85,B 0,C 180,E1 -16460.47,E2 -16460.47} C_VEL
LIN {X 0,Y 297.815,Z 454.042,A -85,B 0,C 180,E1 -16462.645,E2 -16462.645} C_VEL
LIN {X 0,Y 298.621,Z 447.36,A -85,B 0,C 180,E1 -16464.598,E2 -16464.598} C_VEL
LIN {X 0,Y 299.464,Z 440.221,A -85,B 0,C 180,E1 -16466.299,E2 -16466.299} C_VEL
LIN {X 0,Y 300.564,Z 431.57,A -85,B 0,C 180,E1 -16467.99,E2 -16467.99} C_VEL
LIN {X 0,Y 301.868,Z 421.674,A -85,B 0,C 180,E1 -16469.55,E2 -16469.55} C_VEL
LIN {X 0,Y 303.189,Z 410.152,A -85,B 0,C 180,E1 -16471.002,E2 -16471.002} C_VEL
LIN {X 0,Y 304.313,Z 398.433,A -85,B 0,C 180,E1 -16472.15,E2 -16472.15} C_VEL
LIN {X 0,Y 305.199,Z 386.227,A -85,B 0,C 180,E1 -16473.052,E2 -16473.052} C_VEL
LIN {X 0,Y 306.079,Z 372.754,A -85,B 0,C 180,E1 -16473.743,E2 -16473.743} C_VEL
LIN {X 0,Y 306.523,Z 357.789,A -85,B 0,C 180,E1 -16474.191,E2 -16474.191} C_VEL
LIN {X 0,Y 307.962,Z 293.599,A -85,B 0,C 180,E1 -16475.682,E2 -16475.682} C_VEL
LIN {X 0,Y 304.11,Z 271.079,A -85,B 0,C 180,E1 -16476.495,E2 -16476.495} C_VEL
LIN {X 0,Y 300.714,Z 260.333,A -85,B 0,C 180,E1 -16477.047,E2 -16477.047} C_VEL
LIN {X 0,Y 299.713,Z 254.803,A -85,B 0,C 180,E1 -16478.767,E2 -16478.767} C_VEL
LIN {X 0,Y 298.663,Z 249.877,A -85,B 0,C 180,E1 -16480.507,E2 -16480.507} C_VEL
LIN {X 0,Y 298.562,Z 249.791,A -85,B 0,C 180,E1 -16485.211,E2 -16485.211} C_VEL
LIN {X 0,Y 298.523,Z 249.776,A -85,B 0,C 180,E1 -16489.686,E2 -16489.686} C_VEL
LIN {X 0,Y 298.448,Z 249.804,A -85,B 0,C 180,E1 -16493.598,E2 -16493.598} C_VEL
LIN {X 0,Y 298.45,Z 249.769,A -85,B 0,C 180,E1 -16496.577,E2 -16496.577} C_VEL
LIN {X 0,Y 298.423,Z 249.799,A -85,B 0,C 180,E1 -16499.64,E2 -16499.64} C_VEL
LIN {X 0,Y 298.408,Z 249.816,A -85,B 0,C 180,E1 -16502.798,E2 -16502.798} C_VEL
LIN {X 0,Y 298.462,Z 249.8,A -85,B 0,C 180,E1 -16506.825,E2 -16506.825} C_VEL
LIN {X 0,Y 298.439,Z 249.798,A -85,B 0,C 180,E1 -16511.111,E2 -16511.111} C_VEL
LIN {X 0,Y 298.461,Z 249.802,A -85,B 0,C 180,E1 -16515.067,E2 -16515.067} C_VEL
LIN {X 0,Y 298.424,Z 249.802,A -85,B 0,C 180,E1 -16518.903,E2 -16518.903} C_VEL
LIN {X 0,Y 298.397,Z 249.785,A -85,B 0,C 180,E1 -16521.43,E2 -16521.43} C_VEL
LIN {X 0,Y 297.718,Z 249.878,A -85,B 0,C 180,E1 -16522.557,E2 -16522.557} C_VEL
LIN {X 0,Y 294.826,Z 250.252,A -85,B 0,C 180,E1 -16524.392,E2 -16524.392} C_VEL
LIN {X 0,Y 292.395,Z 250.561,A -85,B 0,C 180,E1 -16525.88,E2 -16525.88} C_VEL
LIN {X 0,Y 291.381,Z 250.687,A -85,B 0,C 180,E1 -16527.034,E2 -16527.034} C_VEL
LIN {X 0,Y 291.314,Z 250.694,A -85,B 0,C 180,E1 -16527.425,E2 -16527.425} C_VEL
LIN {X 0,Y 291.361,Z 250.661,A -85,B 0,C 180,E1 -16531.165,E2 -16531.165} C_VEL
LIN {X 0,Y 291.399,Z 250.663,A -85,B 0,C 180,E1 -16534.278,E2 -16534.278} C_VEL
LIN {X 0,Y 291.375,Z 250.689,A -85,B 0,C 180,E1 -16537.307,E2 -16537.307} C_VEL
LIN {X 0,Y 291.489,Z 250.672,A -85,B 0,C 180,E1 -16540.28,E2 -16540.28} C_VEL
LIN {X 0,Y 291.528,Z 250.628,A -85,B 0,C 180,E1 -16544.641,E2 -16544.641} C_VEL
LIN {X 0,Y 291.529,Z 250.66,A -85,B 0,C 180,E1 -16548.887,E2 -16548.887} C_VEL
LIN {X 0,Y 291.702,Z 250.648,A -85,B 0,C 180,E1 -16551.695,E2 -16551.695} C_VEL
LIN {X 0,Y 291.625,Z 250.645,A -85,B 0,C 180,E1 -16554.475,E2 -16554.475} C_VEL
LIN {X 0,Y 291.884,Z 250.588,A -85,B 0,C 180,E1 -16558.627,E2 -16558.627} C_VEL
LIN {X 0,Y 291.886,Z 250.613,A -85,B 0,C 180,E1 -16561.386,E2 -16561.386} C_VEL
LIN {X 0,Y 291.61,Z 250.66,A -85,B 0,C 180,E1 -16565.538,E2 -16565.538} C_VEL
LIN {X 0,Y 291.67,Z 250.626,A -85,B 0,C 180,E1 -16568.918,E2 -16568.918} C_VEL
LIN {X 0,Y 291.521,Z 250.653,A -85,B 0,C 180,E1 -16572.537,E2 -16572.537} C_VEL
LIN {X 0,Y 291.56,Z 250.664,A -85,B 0,C 180,E1 -16575.382,E2 -16575.382} C_VEL
LIN {X 0,Y 291.457,Z 250.658,A -85,B 0,C 180,E1 -16579.88,E2 -16579.88} C_VEL
LIN {X 0,Y 291.389,Z 250.684,A -85,B 0,C 180,E1 -16584.212,E2 -16584.212} C_VEL
LIN {X 0,Y 291.42,Z 250.68,A -85,B 0,C 180,E1 -16587.277,E2 -16587.277} C_VEL
LIN {X 0,Y 291.332,Z 250.675,A -85,B 0,C 180,E1 -16590.443,E2 -16590.443} C_VEL
LIN {X 0,Y 291.353,Z 250.695,A -85,B 0,C 180,E1 -16593.703,E2 -16593.703} C_VEL
LIN {X 0,Y 291.369,Z 250.678,A -85,B 0,C 180,E1 -16597.253,E2 -16597.253} C_VEL
LIN {X 0,Y 291.343,Z 250.694,A -85,B 0,C 180,E1 -16600.647,E2 -16600.647} C_VEL
LIN {X 0,Y 291.303,Z 250.66,A -85,B 0,C 180,E1 -16604.406,E2 -16604.406} C_VEL
LIN {X 0,Y 291.307,Z 250.696,A -85,B 0,C 180,E1 -16608.415,E2 -16608.415} C_VEL
LIN {X 0,Y 291.399,Z 250.679,A -85,B 0,C 180,E1 -16612.919,E2 -16612.919} C_VEL
LIN {X 0,Y 291.357,Z 250.686,A -85,B 0,C 180,E1 -16616.304,E2 -16616.304} C_VEL
LIN {X 0,Y 291.422,Z 250.834,A -85,B 0,C 180,E1 -16619.072,E2 -16619.072} C_VEL
LIN {X 0,Y 293.492,Z 260.739,A -85,B 0,C 180,E1 -16622.384,E2 -16622.384} C_VEL
LIN {X 0,Y 294.747,Z 267.685,A -85,B 0,C 180,E1 -16624.537,E2 -16624.537} C_VEL
LIN {X 0,Y 296.094,Z 272.898,A -85,B 0,C 180,E1 -16624.822,E2 -16624.822} C_VEL
LIN {X 0,Y 301.14,Z 307.878,A -85,B 0,C 180,E1 -16626.065,E2 -16626.065} C_VEL
LIN {X 0,Y 299.506,Z 376.069,A -85,B 0,C 180,E1 -16627.722,E2 -16627.722} C_VEL
LIN {X 0,Y 298.695,Z 389.896,A -85,B 0,C 180,E1 -16628.34,E2 -16628.34} C_VEL
LIN {X 0,Y 297.653,Z 402.323,A -85,B 0,C 180,E1 -16629.168,E2 -16629.168} C_VEL
LIN {X 0,Y 296.451,Z 414.241,A -85,B 0,C 180,E1 -16630.256,E2 -16630.256} C_VEL
LIN {X 0,Y 295.065,Z 425.697,A -85,B 0,C 180,E1 -16631.604,E2 -16631.604} C_VEL
LIN {X 0,Y 293.979,Z 435.159,A -85,B 0,C 180,E1 -16633.003,E2 -16633.003} C_VEL
LIN {X 0,Y 292.793,Z 444.461,A -85,B 0,C 180,E1 -16634.691,E2 -16634.691} C_VEL
LIN {X 0,Y 291.577,Z 453.594,A -85,B 0,C 180,E1 -16636.763,E2 -16636.763} C_VEL
LIN {X 0,Y 290.673,Z 460.941,A -85,B 0,C 180,E1 -16638.848,E2 -16638.848} C_VEL
LIN {X 0,Y 290.038,Z 466.806,A -85,B 0,C 180,E1 -16640.938,E2 -16640.938} C_VEL
LIN {X 0,Y 289.623,Z 471.404,A -85,B 0,C 180,E1 -16643.032,E2 -16643.032} C_VEL
LIN {X 0,Y 289.444,Z 474.106,A -85,B 0,C 180,E1 -16644.614,E2 -16644.614} C_VEL
LIN {X 0,Y 289.401,Z 477.351,A -85,B 0,C 180,E1 -16647.217,E2 -16647.217} C_VEL
LIN {X 0,Y 289.382,Z 478.46,A -85,B 0,C 180,E1 -16648.609,E2 -16648.609} C_VEL
LIN {X 0,Y 289.382,Z 479.153,A -85,B 0,C 180,E1 -16650,E2 -16650} C_VEL
LIN {X 0,Y 289.382,Z 479.459,A -85,B 0,C 180,E1 -16651.392,E2 -16651.392} C_VEL
LIN {X 0,Y 289.405,Z 479.382,A -85,B 0,C 180,E1 -16652.784,E2 -16652.784} C_VEL
LIN {X 0,Y 289.426,Z 478.896,A -85,B 0,C 180,E1 -16654.178,E2 -16654.178} C_VEL
LIN {X 0,Y 289.73,Z 476.706,A -85,B 0,C 180,E1 -16656.967,E2 -16656.967} C_VEL
LIN {X 0,Y 290.265,Z 473.991,A -85,B 0,C 180,E1 -16659.055,E2 -16659.055} C_VEL
LIN {X 0,Y 291.084,Z 470.278,A -85,B 0,C 180,E1 -16661.137,E2 -16661.137} C_VEL
LIN {X 0,Y 292.185,Z 465.472,A -85,B 0,C 180,E1 -16663.21,E2 -16663.21} C_VEL
LIN {X 0,Y 293.661,Z 459.435,A -85,B 0,C 180,E1 -16665.264,E2 -16665.264} C_VEL
LIN {X 0,Y 295.524,Z 451.948,A -85,B 0,C 180,E1 -16667.294,E2 -16667.294} C_VEL
LIN {X 0,Y 297.173,Z 444.149,A -85,B 0,C 180,E1 -16669.018,E2 -16669.018} C_VEL
LIN {X 0,Y 299.379,Z 434.033,A -85,B 0,C 180,E1 -16670.798,E2 -16670.798} C_VEL
LIN {X 0,Y 301.524,Z 423.558,A -85,B 0,C 180,E1 -16672.257,E2 -16672.257} C_VEL
LIN {X 0,Y 303.543,Z 411.902,A -85,B 0,C 180,E1 -16673.541,E2 -16673.541} C_VEL
LIN {X 0,Y 305.377,Z 399.452,A -85,B 0,C 180,E1 -16674.563,E2 -16674.563} C_VEL
LIN {X 0,Y 306.766,Z 387.123,A -85,B 0,C 180,E1 -16675.304,E2 -16675.304} C_VEL
LIN {X 0,Y 307.713,Z 374.357,A -85,B 0,C 180,E1 -16675.82,E2 -16675.82} C_VEL
LIN {X 0,Y 309.78,Z 310.247,A -85,B 0,C 180,E1 -16677.364,E2 -16677.364} C_VEL
LIN {X 0,Y 306.786,Z 293.948,A -85,B 0,C 180,E1 -16678.175,E2 -16678.175} C_VEL
LIN {X 0,Y 305.38,Z 288.134,A -85,B 0,C 180,E1 -16678.513,E2 -16678.513} C_VEL
LIN {X 0,Y 299.165,Z 274.606,A -85,B 0,C 180,E1 -16679.708,E2 -16679.708} C_VEL
LIN {X 0,Y 295.539,Z 267.207,A -85,B 0,C 180,E1 -16680.468,E2 -16680.468} C_VEL
LIN {X 0,Y 293.786,Z 259.959,A -85,B 0,C 180,E1 -16683.139,E2 -16683.139} C_VEL
LIN {X 0,Y 291.895,Z 252.508,A -85,B 0,C 180,E1 -16686.15,E2 -16686.15} C_VEL
LIN {X 0,Y 291.404,Z 250.715,A -85,B 0,C 180,E1 -16687.027,E2 -16687.027} C_VEL
LIN {X 0,Y 291.316,Z 250.7,A -85,B 0,C 180,E1 -16690.646,E2 -16690.646} C_VEL
LIN {X 0,Y 291.298,Z 250.698,A -85,B 0,C 180,E1 -16694.401,E2 -16694.401} C_VEL
LIN {X 0,Y 291.332,Z 250.678,A -85,B 0,C 180,E1 -16698.404,E2 -16698.404} C_VEL
LIN {X 0,Y 291.353,Z 250.687,A -85,B 0,C 180,E1 -16701.152,E2 -16701.152} C_VEL
LIN {X 0,Y 291.369,Z 250.685,A -85,B 0,C 180,E1 -16704.621,E2 -16704.621} C_VEL
LIN {X 0,Y 291.378,Z 250.681,A -85,B 0,C 180,E1 -16707.946,E2 -16707.946} C_VEL
LIN {X 0,Y 291.354,Z 250.685,A -85,B 0,C 180,E1 -16711.15,E2 -16711.15} C_VEL
LIN {X 0,Y 291.354,Z 250.692,A -85,B 0,C 180,E1 -16714.26,E2 -16714.26} C_VEL
LIN {X 0,Y 291.364,Z 250.69,A -85,B 0,C 180,E1 -16717.292,E2 -16717.292} C_VEL
LIN {X 0,Y 291.399,Z 250.675,A -85,B 0,C 180,E1 -16720.26,E2 -16720.26} C_VEL
LIN {X 0,Y 291.506,Z 250.66,A -85,B 0,C 180,E1 -16724.66,E2 -16724.66} C_VEL
LIN {X 0,Y 291.536,Z 250.659,A -85,B 0,C 180,E1 -16728.875,E2 -16728.875} C_VEL
LIN {X 0,Y 291.667,Z 250.656,A -85,B 0,C 180,E1 -16731.681,E2 -16731.681} C_VEL
LIN {X 0,Y 291.611,Z 250.651,A -85,B 0,C 180,E1 -16734.462,E2 -16734.462} C_VEL
LIN {X 0,Y 291.884,Z 250.615,A -85,B 0,C 180,E1 -16738.614,E2 -16738.614} C_VEL
LIN {X 0,Y 291.884,Z 250.626,A -85,B 0,C 180,E1 -16741.373,E2 -16741.373} C_VEL
LIN {X 0,Y 291.691,Z 250.64,A -85,B 0,C 180,E1 -16746.913,E2 -16746.913} C_VEL
LIN {X 0,Y 291.568,Z 250.666,A -85,B 0,C 180,E1 -16749.707,E2 -16749.707} C_VEL
LIN {X 0,Y 291.508,Z 250.674,A -85,B 0,C 180,E1 -16753.944,E2 -16753.944} C_VEL
LIN {X 0,Y 291.438,Z 250.678,A -85,B 0,C 180,E1 -16758.262,E2 -16758.262} C_VEL
LIN {X 0,Y 291.361,Z 250.688,A -85,B 0,C 180,E1 -16761.204,E2 -16761.204} C_VEL
LIN {X 0,Y 291.385,Z 250.686,A -85,B 0,C 180,E1 -16764.199,E2 -16764.199} C_VEL
LIN {X 0,Y 291.399,Z 250.669,A -85,B 0,C 180,E1 -16767.266,E2 -16767.266} C_VEL
LIN {X 0,Y 291.315,Z 250.683,A -85,B 0,C 180,E1 -16770.431,E2 -16770.431} C_VEL
LIN {X 0,Y 291.324,Z 250.694,A -85,B 0,C 180,E1 -16773.692,E2 -16773.692} C_VEL
LIN {X 0,Y 291.436,Z 250.891,A -85,B 0,C 180,E1 -16777.446,E2 -16777.446} C_VEL
LIN {X 0,Y 293.794,Z 259.837,A -85,B 0,C 180,E1 -16781.125,E2 -16781.125} C_VEL
LIN {X 0,Y 294.178,Z 260.946,A -85,B 0,C 180,E1 -16781.401,E2 -16781.401} C_VEL
LIN {X 0,Y 302.702,Z 277.691,A -85,B 0,C 180,E1 -16783.083,E2 -16783.083} C_VEL
LIN {X 0,Y 308.649,Z 291.151,A -85,B 0,C 180,E1 -16784.21,E2 -16784.21} C_VEL
LIN {X 0,Y 310.242,Z 299.734,A -85,B 0,C 180,E1 -16784.637,E2 -16784.637} C_VEL
LIN {X 0,Y 307.774,Z 368.458,A -85,B 0,C 180,E1 -16786.281,E2 -16786.281} C_VEL
LIN {X 0,Y 306.702,Z 382.114,A -85,B 0,C 180,E1 -16786.873,E2 -16786.873} C_VEL
LIN {X 0,Y 305.278,Z 394.97,A -85,B 0,C 180,E1 -16787.712,E2 -16787.712} C_VEL
LIN {X 0,Y 303.616,Z 406.347,A -85,B 0,C 180,E1 -16788.722,E2 -16788.722} C_VEL
LIN {X 0,Y 301.601,Z 418.197,A -85,B 0,C 180,E1 -16790.091,E2 -16790.091} C_VEL
LIN {X 0,Y 299.594,Z 428.259,A -85,B 0,C 180,E1 -16791.563,E2 -16791.563} C_VEL
LIN {X 0,Y 297.525,Z 437.671,A -85,B 0,C 180,E1 -16793.293,E2 -16793.293} C_VEL
LIN {X 0,Y 295.572,Z 446.025,A -85,B 0,C 180,E1 -16795.203,E2 -16795.203} C_VEL
LIN {X 0,Y 293.593,Z 453.803,A -85,B 0,C 180,E1 -16797.439,E2 -16797.439} C_VEL
LIN {X 0,Y 292.109,Z 459.735,A -85,B 0,C 180,E1 -16799.652,E2 -16799.652} C_VEL
LIN {X 0,Y 290.959,Z 464.366,A -85,B 0,C 180,E1 -16801.899,E2 -16801.899} C_VEL
LIN {X 0,Y 290.172,Z 467.767,A -85,B 0,C 180,E1 -16804.153,E2 -16804.153} C_VEL
LIN {X 0,Y 289.767,Z 469.421,A -85,B 0,C 180,E1 -16805.649,E2 -16805.649} C_VEL
LIN {X 0,Y 289.47,Z 470.643,A -85,B 0,C 180,E1 -16807.286,E2 -16807.286} C_VEL
LIN {X 0,Y 289.141,Z 471.52,A -85,B 0,C 180,E1 -16810.105,E2 -16810.105} C_VEL
LIN {X 0,Y 289.11,Z 471.32,A -85,B 0,C 180,E1 -16811.577,E2 -16811.577} C_VEL
LIN {X 0,Y 289.07,Z 470.68,A -85,B 0,C 180,E1 -16813.037,E2 -16813.037} C_VEL
LIN {X 0,Y 289.152,Z 469.627,A -85,B 0,C 180,E1 -16814.492,E2 -16814.492} C_VEL
LIN {X 0,Y 289.32,Z 467.678,A -85,B 0,C 180,E1 -16816.289,E2 -16816.289} C_VEL
LIN {X 0,Y 289.722,Z 463.736,A -85,B 0,C 180,E1 -16818.81,E2 -16818.81} C_VEL
LIN {X 0,Y 290.167,Z 459.162,A -85,B 0,C 180,E1 -16820.942,E2 -16820.942} C_VEL
LIN {X 0,Y 290.887,Z 453.33,A -85,B 0,C 180,E1 -16823.061,E2 -16823.061} C_VEL
LIN {X 0,Y 291.784,Z 446.01,A -85,B 0,C 180,E1 -16825.164,E2 -16825.164} C_VEL
LIN {X 0,Y 292.951,Z 436.915,A -85,B 0,C 180,E1 -16827.249,E2 -16827.249} C_VEL
LIN {X 0,Y 294.179,Z 427.525,A -85,B 0,C 180,E1 -16828.973,E2 -16828.973} C_VEL
LIN {X 0,Y 295.585,Z 416.7,A -85,B 0,C 180,E1 -16830.552,E2 -16830.552} C_VEL
LIN {X 0,Y 296.813,Z 405.384,A -85,B 0,C 180,E1 -16831.865,E2 -16831.865} C_VEL
LIN {X 0,Y 297.941,Z 393.105,A -85,B 0,C 180,E1 -16832.957,E2 -16832.957} C_VEL
LIN {X 0,Y 298.825,Z 380.938,A -85,B 0,C 180,E1 -16833.75,E2 -16833.75} C_VEL
LIN {X 0,Y 299.519,Z 367.718,A -85,B 0,C 180,E1 -16834.331,E2 -16834.331} C_VEL
LIN {X 0,Y 301.23,Z 294.414,A -85,B 0,C 180,E1 -16836.102,E2 -16836.102} C_VEL
LIN {X 0,Y 297.551,Z 272.932,A -85,B 0,C 180,E1 -16836.901,E2 -16836.901} C_VEL
LIN {X 0,Y 293.503,Z 260.336,A -85,B 0,C 180,E1 -16837.569,E2 -16837.569} C_VEL
LIN {X 0,Y 291.828,Z 251.82,A -85,B 0,C 180,E1 -16840.405,E2 -16840.405} C_VEL
LIN {X 0,Y 291.566,Z 250.689,A -85,B 0,C 180,E1 -16840.942,E2 -16840.942} C_VEL
LIN {X 0,Y 291.512,Z 250.67,A -85,B 0,C 180,E1 -16845.378,E2 -16845.378} C_VEL
LIN {X 0,Y 291.454,Z 250.657,A -85,B 0,C 180,E1 -16849.902,E2 -16849.902} C_VEL
LIN {X 0,Y 291.397,Z 250.678,A -85,B 0,C 180,E1 -16854.205,E2 -16854.205} C_VEL
LIN {X 0,Y 291.387,Z 250.648,A -85,B 0,C 180,E1 -16857.274,E2 -16857.274} C_VEL
LIN {X 0,Y 291.359,Z 250.688,A -85,B 0,C 180,E1 -16860.434,E2 -16860.434} C_VEL
LIN {X 0,Y 291.358,Z 250.686,A -85,B 0,C 180,E1 -16863.696,E2 -16863.696} C_VEL
LIN {X 0,Y 291.426,Z 250.679,A -85,B 0,C 180,E1 -16867.28,E2 -16867.28} C_VEL
LIN {X 0,Y 291.39,Z 250.679,A -85,B 0,C 180,E1 -16870.632,E2 -16870.632} C_VEL
LIN {X 0,Y 291.382,Z 250.682,A -85,B 0,C 180,E1 -16874.383,E2 -16874.383} C_VEL
LIN {X 0,Y 291.36,Z 250.684,A -85,B 0,C 180,E1 -16878.396,E2 -16878.396} C_VEL
LIN {X 0,Y 291.346,Z 250.663,A -85,B 0,C 180,E1 -16881.421,E2 -16881.421} C_VEL
LIN {X 0,Y 291.365,Z 250.687,A -85,B 0,C 180,E1 -16885.095,E2 -16885.095} C_VEL
LIN {X 0,Y 291.314,Z 250.694,A -85,B 0,C 180,E1 -16887.425,E2 -16887.425} C_VEL
LIN {X 0,Y 290.693,Z 250.769,A -85,B 0,C 180,E1 -16888.579,E2 -16888.579} C_VEL
LIN {X 0,Y 287.875,Z 251.102,A -85,B 0,C 180,E1 -16890.458,E2 -16890.458} C_VEL
LIN {X 0,Y 285.466,Z 251.39,A -85,B 0,C 180,E1 -16891.983,E2 -16891.983} C_VEL
LIN {X 0,Y 284.438,Z 251.52,A -85,B 0,C 180,E1 -16893.164,E2 -16893.164} C_VEL
LIN {X 0,Y 284.359,Z 251.534,A -85,B 0,C 180,E1 -16893.565,E2 -16893.565} C_VEL
LIN {X 0,Y 284.353,Z 251.56,A -85,B 0,C 180,E1 -16896.714,E2 -16896.714} C_VEL
LIN {X 0,Y 284.416,Z 251.552,A -85,B 0,C 180,E1 -16899.881,E2 -16899.881} C_VEL
LIN {X 0,Y 284.466,Z 251.507,A -85,B 0,C 180,E1 -16904.476,E2 -16904.476} C_VEL
LIN {X 0,Y 284.481,Z 251.536,A -85,B 0,C 180,E1 -16908.608,E2 -16908.608} C_VEL
LIN {X 0,Y 284.652,Z 251.528,A -85,B 0,C 180,E1 -16911.488,E2 -16911.488} C_VEL
LIN {X 0,Y 284.596,Z 251.521,A -85,B 0,C 180,E1 -16914.338,E2 -16914.338} C_VEL
LIN {X 0,Y 284.851,Z 251.462,A -85,B 0,C 180,E1 -16918.593,E2 -16918.593} C_VEL
LIN {X 0,Y 284.852,Z 251.489,A -85,B 0,C 180,E1 -16921.42,E2 -16921.42} C_VEL
LIN {X 0,Y 284.579,Z 251.535,A -85,B 0,C 180,E1 -16925.675,E2 -16925.675} C_VEL
LIN {X 0,Y 284.611,Z 251.503,A -85,B 0,C 180,E1 -16928.989,E2 -16928.989} C_VEL
LIN {X 0,Y 284.478,Z 251.535,A -85,B 0,C 180,E1 -16932.853,E2 -16932.853} C_VEL
LIN {X 0,Y 284.492,Z 251.546,A -85,B 0,C 180,E1 -16935.774,E2 -16935.774} C_VEL
LIN {X 0,Y 284.384,Z 251.534,A -85,B 0,C 180,E1 -16940.248,E2 -16940.248} C_VEL
LIN {X 0,Y 284.343,Z 251.568,A -85,B 0,C 180,E1 -16944.852,E2 -16944.852} C_VEL
LIN {X 0,Y 284.326,Z 251.563,A -85,B 0,C 180,E1 -16948.017,E2 -16948.017} C_VEL
LIN {X 0,Y 284.296,Z 251.56,A -85,B 0,C 180,E1 -16951.28,E2 -16951.28} C_VEL
LIN {X 0,Y 284.347,Z 251.561,A -85,B 0,C 180,E1 -16955.351,E2 -16955.351} C_VEL
LIN {X 0,Y 284.313,Z 251.562,A -85,B 0,C 180,E1 -16958.175,E2 -16958.175} C_VEL
LIN {X 0,Y 284.281,Z 251.564,A -85,B 0,C 180,E1 -16962.128,E2 -16962.128} C_VEL
LIN {X 0,Y 284.249,Z 251.54,A -85,B 0,C 180,E1 -16966.189,E2 -16966.189} C_VEL
LIN {X 0,Y 284.269,Z 251.573,A -85,B 0,C 180,E1 -16970.04,E2 -16970.04} C_VEL
LIN {X 0,Y 284.332,Z 251.566,A -85,B 0,C 180,E1 -16973.615,E2 -16973.615} C_VEL
LIN {X 0,Y 284.335,Z 251.565,A -85,B 0,C 180,E1 -16977.899,E2 -16977.899} C_VEL
LIN {X 0,Y 284.366,Z 251.776,A -85,B 0,C 180,E1 -16978.735,E2 -16978.735} C_VEL
LIN {X 0,Y 286.527,Z 261.949,A -85,B 0,C 180,E1 -16982.223,E2 -16982.223} C_VEL
LIN {X 0,Y 287.587,Z 267.785,A -85,B 0,C 180,E1 -16984.029,E2 -16984.029} C_VEL
LIN {X 0,Y 289.543,Z 274.578,A -85,B 0,C 180,E1 -16984.396,E2 -16984.396} C_VEL
LIN {X 0,Y 294.402,Z 308.044,A -85,B 0,C 180,E1 -16985.614,E2 -16985.614} C_VEL
LIN {X 0,Y 292.773,Z 375.466,A -85,B 0,C 180,E1 -16987.286,E2 -16987.286} C_VEL
LIN {X 0,Y 292.009,Z 388.515,A -85,B 0,C 180,E1 -16987.864,E2 -16987.864} C_VEL
LIN {X 0,Y 291.019,Z 400.75,A -85,B 0,C 180,E1 -16988.67,E2 -16988.67} C_VEL
LIN {X 0,Y 289.743,Z 413.084,A -85,B 0,C 180,E1 -16989.779,E2 -16989.779} C_VEL
LIN {X 0,Y 288.232,Z 424.727,A -85,B 0,C 180,E1 -16991.151,E2 -16991.151} C_VEL
LIN {X 0,Y 287,Z 435.442,A -85,B 0,C 180,E1 -16992.763,E2 -16992.763} C_VEL
LIN {X 0,Y 285.93,Z 443.801,A -85,B 0,C 180,E1 -16994.314,E2 -16994.314} C_VEL
LIN {X 0,Y 284.633,Z 453.044,A -85,B 0,C 180,E1 -16996.434,E2 -16996.434} C_VEL
LIN {X 0,Y 283.647,Z 460.468,A -85,B 0,C 180,E1 -16998.568,E2 -16998.568} C_VEL
LIN {X 0,Y 282.985,Z 466.41,A -85,B 0,C 180,E1 -17000.711,E2 -17000.711} C_VEL
LIN {X 0,Y 282.571,Z 471.079,A -85,B 0,C 180,E1 -17002.857,E2 -17002.857} C_VEL
LIN {X 0,Y 282.351,Z 474.146,A -85,B 0,C 180,E1 -17004.689,E2 -17004.689} C_VEL
LIN {X 0,Y 282.31,Z 477.133,A -85,B 0,C 180,E1 -17007.147,E2 -17007.147} C_VEL
LIN {X 0,Y 282.307,Z 478.295,A -85,B 0,C 180,E1 -17008.574,E2 -17008.574} C_VEL
LIN {X 0,Y 282.305,Z 479.015,A -85,B 0,C 180,E1 -17010,E2 -17010} C_VEL
LIN {X 0,Y 282.307,Z 479.348,A -85,B 0,C 180,E1 -17011.427,E2 -17011.427} C_VEL
LIN {X 0,Y 282.316,Z 479.296,A -85,B 0,C 180,E1 -17012.854,E2 -17012.854} C_VEL
LIN {X 0,Y 282.441,Z 478.151,A -85,B 0,C 180,E1 -17015.506,E2 -17015.506} C_VEL
LIN {X 0,Y 282.68,Z 476.729,A -85,B 0,C 180,E1 -17017.141,E2 -17017.141} C_VEL
LIN {X 0,Y 283.256,Z 474.074,A -85,B 0,C 180,E1 -17019.281,E2 -17019.281} C_VEL
LIN {X 0,Y 284.094,Z 470.426,A -85,B 0,C 180,E1 -17021.415,E2 -17021.415} C_VEL
LIN {X 0,Y 285.249,Z 465.692,A -85,B 0,C 180,E1 -17023.537,E2 -17023.537} C_VEL
LIN {X 0,Y 286.823,Z 459.728,A -85,B 0,C 180,E1 -17025.637,E2 -17025.637} C_VEL
LIN {X 0,Y 288.758,Z 452.323,A -85,B 0,C 180,E1 -17027.712,E2 -17027.712} C_VEL
LIN {X 0,Y 290.819,Z 443.137,A -85,B 0,C 180,E1 -17029.775,E2 -17029.775} C_VEL
LIN {X 0,Y 293.07,Z 433.614,A -85,B 0,C 180,E1 -17031.451,E2 -17031.451} C_VEL
LIN {X 0,Y 295.248,Z 423.08,A -85,B 0,C 180,E1 -17032.942,E2 -17032.942} C_VEL
LIN {X 0,Y 297.11,Z 412.928,A -85,B 0,C 180,E1 -17034.082,E2 -17034.082} C_VEL
LIN {X 0,Y 299.016,Z 400.909,A -85,B 0,C 180,E1 -17035.122,E2 -17035.122} C_VEL
LIN {X 0,Y 300.514,Z 388.371,A -85,B 0,C 180,E1 -17035.915,E2 -17035.915} C_VEL
LIN {X 0,Y 301.594,Z 375.116,A -85,B 0,C 180,E1 -17036.482,E2 -17036.482} C_VEL
LIN {X 0,Y 303.778,Z 311.217,A -85,B 0,C 180,E1 -17038.058,E2 -17038.058} C_VEL
LIN {X 0,Y 300.756,Z 294.956,A -85,B 0,C 180,E1 -17038.907,E2 -17038.907} C_VEL
LIN {X 0,Y 299.777,Z 291.022,A -85,B 0,C 180,E1 -17039.148,E2 -17039.148} C_VEL
LIN {X 0,Y 293.234,Z 276.849,A -85,B 0,C 180,E1 -17040.459,E2 -17040.459} C_VEL
LIN {X 0,Y 288.304,Z 267.048,A -85,B 0,C 180,E1 -17041.531,E2 -17041.531} C_VEL
LIN {X 0,Y 286.2,Z 258.533,A -85,B 0,C 180,E1 -17044.849,E2 -17044.849} C_VEL
LIN {X 0,Y 284.362,Z 251.902,A -85,B 0,C 180,E1 -17047.725,E2 -17047.725} C_VEL
LIN {X 0,Y 284.31,Z 251.559,A -85,B 0,C 180,E1 -17048.17,E2 -17048.17} C_VEL
LIN {X 0,Y 284.252,Z 251.562,A -85,B 0,C 180,E1 -17052.114,E2 -17052.114} C_VEL
LIN {X 0,Y 284.271,Z 251.559,A -85,B 0,C 180,E1 -17056.186,E2 -17056.186} C_VEL
LIN {X 0,Y 284.321,Z 251.57,A -85,B 0,C 180,E1 -17060.021,E2 -17060.021} C_VEL
LIN {X 0,Y 284.334,Z 251.566,A -85,B 0,C 180,E1 -17063.608,E2 -17063.608} C_VEL
LIN {X 0,Y 284.319,Z 251.564,A -85,B 0,C 180,E1 -17067.186,E2 -17067.186} C_VEL
LIN {X 0,Y 284.349,Z 251.566,A -85,B 0,C 180,E1 -17070.369,E2 -17070.369} C_VEL
LIN {X 0,Y 284.309,Z 251.571,A -85,B 0,C 180,E1 -17073.574,E2 -17073.574} C_VEL
LIN {X 0,Y 284.319,Z 251.562,A -85,B 0,C 180,E1 -17076.697,E2 -17076.697} C_VEL
LIN {X 0,Y 284.342,Z 251.56,A -85,B 0,C 180,E1 -17081.252,E2 -17081.252} C_VEL
LIN {X 0,Y 284.472,Z 251.543,A -85,B 0,C 180,E1 -17085.691,E2 -17085.691} C_VEL
LIN {X 0,Y 284.52,Z 251.536,A -85,B 0,C 180,E1 -17090.037,E2 -17090.037} C_VEL
LIN {X 0,Y 284.658,Z 251.52,A -85,B 0,C 180,E1 -17092.903,E2 -17092.903} C_VEL
LIN {X 0,Y 284.85,Z 251.491,A -85,B 0,C 180,E1 -17098.58,E2 -17098.58} C_VEL
LIN {X 0,Y 284.85,Z 251.503,A -85,B 0,C 180,E1 -17101.407,E2 -17101.407} C_VEL
LIN {X 0,Y 284.646,Z 251.517,A -85,B 0,C 180,E1 -17107.085,E2 -17107.085} C_VEL
LIN {X 0,Y 284.513,Z 251.546,A -85,B 0,C 180,E1 -17109.95,E2 -17109.95} C_VEL
LIN {X 0,Y 284.456,Z 251.548,A -85,B 0,C 180,E1 -17114.297,E2 -17114.297} C_VEL
LIN {X 0,Y 284.375,Z 251.556,A -85,B 0,C 180,E1 -17118.733,E2 -17118.733} C_VEL
LIN {X 0,Y 284.353,Z 251.567,A -85,B 0,C 180,E1 -17123.286,E2 -17123.286} C_VEL
LIN {X 0,Y 284.376,Z 251.542,A -85,B 0,C 180,E1 -17127.165,E2 -17127.165} C_VEL
LIN {X 0,Y 284.274,Z 251.557,A -85,B 0,C 180,E1 -17131.268,E2 -17131.268} C_VEL
LIN {X 0,Y 284.341,Z 251.554,A -85,B 0,C 180,E1 -17135.347,E2 -17135.347} C_VEL
LIN {X 0,Y 284.362,Z 251.795,A -85,B 0,C 180,E1 -17136.53,E2 -17136.53} C_VEL
LIN {X 0,Y 286.766,Z 260.558,A -85,B 0,C 180,E1 -17140.243,E2 -17140.243} C_VEL
LIN {X 0,Y 289.044,Z 264.876,A -85,B 0,C 180,E1 -17140.796,E2 -17140.796} C_VEL
LIN {X 0,Y 297.139,Z 280.653,A -85,B 0,C 180,E1 -17142.432,E2 -17142.432} C_VEL
LIN {X 0,Y 303.027,Z 294.033,A -85,B 0,C 180,E1 -17143.593,E2 -17143.593} C_VEL
LIN {X 0,Y 304.241,Z 300.56,A -85,B 0,C 180,E1 -17143.932,E2 -17143.932} C_VEL
LIN {X 0,Y 301.727,Z 368.473,A -85,B 0,C 180,E1 -17145.591,E2 -17145.591} C_VEL
LIN {X 0,Y 300.581,Z 382.253,A -85,B 0,C 180,E1 -17146.195,E2 -17146.195} C_VEL
LIN {X 0,Y 299.108,Z 395.063,A -85,B 0,C 180,E1 -17147.047,E2 -17147.047} C_VEL
LIN {X 0,Y 297.312,Z 406.748,A -85,B 0,C 180,E1 -17148.103,E2 -17148.103} C_VEL
LIN {X 0,Y 295.226,Z 418.512,A -85,B 0,C 180,E1 -17149.494,E2 -17149.494} C_VEL
LIN {X 0,Y 293.122,Z 428.545,A -85,B 0,C 180,E1 -17150.995,E2 -17150.995} C_VEL
LIN {X 0,Y 290.858,Z 438.299,A -85,B 0,C 180,E1 -17152.837,E2 -17152.837} C_VEL
LIN {X 0,Y 288.881,Z 446.244,A -85,B 0,C 180,E1 -17154.704,E2 -17154.704} C_VEL
LIN {X 0,Y 286.977,Z 453.355,A -85,B 0,C 180,E1 -17156.776,E2 -17156.776} C_VEL
LIN {X 0,Y 285.49,Z 459.034,A -85,B 0,C 180,E1 -17158.871,E2 -17158.871} C_VEL
LIN {X 0,Y 284.202,Z 463.856,A -85,B 0,C 180,E1 -17161.17,E2 -17161.17} C_VEL
LIN {X 0,Y 283.294,Z 467.428,A -85,B 0,C 180,E1 -17163.477,E2 -17163.477} C_VEL
LIN {X 0,Y 282.816,Z 469.165,A -85,B 0,C 180,E1 -17165.01,E2 -17165.01} C_VEL
LIN {X 0,Y 282.408,Z 470.728,A -85,B 0,C 180,E1 -17167.018,E2 -17167.018} C_VEL
LIN {X 0,Y 282.061,Z 471.583,A -85,B 0,C 180,E1 -17169.584,E2 -17169.584} C_VEL
LIN {X 0,Y 282.019,Z 471.488,A -85,B 0,C 180,E1 -17171.23,E2 -17171.23} C_VEL
LIN {X 0,Y 281.985,Z 470.976,A -85,B 0,C 180,E1 -17172.597,E2 -17172.597} C_VEL
LIN {X 0,Y 282.023,Z 470.001,A -85,B 0,C 180,E1 -17174.09,E2 -17174.09} C_VEL
LIN {X 0,Y 282.223,Z 467.906,A -85,B 0,C 180,E1 -17176.175,E2 -17176.175} C_VEL
LIN {X 0,Y 282.588,Z 464.427,A -85,B 0,C 180,E1 -17178.523,E2 -17178.523} C_VEL
LIN {X 0,Y 283.018,Z 460.026,A -85,B 0,C 180,E1 -17180.711,E2 -17180.711} C_VEL
LIN {X 0,Y 283.687,Z 454.399,A -85,B 0,C 180,E1 -17182.884,E2 -17182.884} C_VEL
LIN {X 0,Y 284.616,Z 447.366,A -85,B 0,C 180,E1 -17185.042,E2 -17185.042} C_VEL
LIN {X 0,Y 285.737,Z 438.55,A -85,B 0,C 180,E1 -17187.18,E2 -17187.18} C_VEL
LIN {X 0,Y 287.155,Z 428.488,A -85,B 0,C 180,E1 -17189.123,E2 -17189.123} C_VEL
LIN {X 0,Y 288.532,Z 418.281,A -85,B 0,C 180,E1 -17190.689,E2 -17190.689} C_VEL
LIN {X 0,Y 289.83,Z 406.822,A -85,B 0,C 180,E1 -17192.084,E2 -17192.084} C_VEL
LIN {X 0,Y 290.993,Z 395.006,A -85,B 0,C 180,E1 -17193.201,E2 -17193.201} C_VEL
LIN {X 0,Y 291.945,Z 382.092,A -85,B 0,C 180,E1 -17194.098,E2 -17194.098} C_VEL
LIN {X 0,Y 292.752,Z 368.196,A -85,B 0,C 180,E1 -17194.733,E2 -17194.733} C_VEL
LIN {X 0,Y 294.514,Z 295.168,A -85,B 0,C 180,E1 -17196.542,E2 -17196.542} C_VEL
LIN {X 0,Y 291.127,Z 275.109,A -85,B 0,C 180,E1 -17197.309,E2 -17197.309} C_VEL
LIN {X 0,Y 286.316,Z 260.375,A -85,B 0,C 180,E1 -17198.113,E2 -17198.113} C_VEL
LIN {X 0,Y 284.546,Z 251.752,A -85,B 0,C 180,E1 -17201.125,E2 -17201.125} C_VEL
LIN {X 0,Y 284.451,Z 251.551,A -85,B 0,C 180,E1 -17205.544,E2 -17205.544} C_VEL
LIN {X 0,Y 284.386,Z 251.54,A -85,B 0,C 180,E1 -17210.241,E2 -17210.241} C_VEL
LIN {X 0,Y 284.36,Z 251.558,A -85,B 0,C 180,E1 -17213.893,E2 -17213.893} C_VEL
LIN {X 0,Y 284.335,Z 251.531,A -85,B 0,C 180,E1 -17218.01,E2 -17218.01} C_VEL
LIN {X 0,Y 284.327,Z 251.569,A -85,B 0,C 180,E1 -17221.27,E2 -17221.27} C_VEL
LIN {X 0,Y 284.358,Z 251.55,A -85,B 0,C 180,E1 -17225.368,E2 -17225.368} C_VEL
LIN {X 0,Y 284.337,Z 251.567,A -85,B 0,C 180,E1 -17228.164,E2 -17228.164} C_VEL
LIN {X 0,Y 284.333,Z 251.545,A -85,B 0,C 180,E1 -17232.151,E2 -17232.151} C_VEL
LIN {X 0,Y 284.326,Z 251.569,A -85,B 0,C 180,E1 -17236.214,E2 -17236.214} C_VEL
LIN {X 0,Y 284.323,Z 251.545,A -85,B 0,C 180,E1 -17240.019,E2 -17240.019} C_VEL
LIN {X 0,Y 284.329,Z 251.553,A -85,B 0,C 180,E1 -17243.624,E2 -17243.624} C_VEL
LIN {X 0,Y 284.272,Z 251.57,A -85,B 0,C 180,E1 -17247.41,E2 -17247.41} C_VEL
LIN {X 0,Y 284.338,Z 251.542,A -85,B 0,C 180,E1 -17250.383,E2 -17250.383} C_VEL
LIN {X 0,Y 284.359,Z 251.534,A -85,B 0,C 180,E1 -17253.565,E2 -17253.565} C_VEL
LIN {X 0,Y 283.712,Z 251.629,A -85,B 0,C 180,E1 -17254.747,E2 -17254.747} C_VEL
LIN {X 0,Y 280.895,Z 251.996,A -85,B 0,C 180,E1 -17256.674,E2 -17256.674} C_VEL
LIN {X 0,Y 278.487,Z 252.297,A -85,B 0,C 180,E1 -17258.238,E2 -17258.238} C_VEL
LIN {X 0,Y 277.441,Z 252.422,A -85,B 0,C 180,E1 -17259.45,E2 -17259.45} C_VEL
LIN {X 0,Y 277.349,Z 252.431,A -85,B 0,C 180,E1 -17259.861,E2 -17259.861} C_VEL
LIN {X 0,Y 277.423,Z 252.384,A -85,B 0,C 180,E1 -17264.29,E2 -17264.29} C_VEL
LIN {X 0,Y 277.427,Z 252.414,A -85,B 0,C 180,E1 -17268.315,E2 -17268.315} C_VEL
LIN {X 0,Y 277.608,Z 252.406,A -85,B 0,C 180,E1 -17271.27,E2 -17271.27} C_VEL
LIN {X 0,Y 277.566,Z 252.397,A -85,B 0,C 180,E1 -17274.194,E2 -17274.194} C_VEL
LIN {X 0,Y 277.817,Z 252.337,A -85,B 0,C 180,E1 -17278.557,E2 -17278.557} C_VEL
LIN {X 0,Y 277.818,Z 252.366,A -85,B 0,C 180,E1 -17281.456,E2 -17281.456} C_VEL
LIN {X 0,Y 277.606,Z 252.393,A -85,B 0,C 180,E1 -17287.278,E2 -17287.278} C_VEL
LIN {X 0,Y 277.459,Z 252.385,A -85,B 0,C 180,E1 -17290.219,E2 -17290.219} C_VEL
LIN {X 0,Y 277.439,Z 252.425,A -85,B 0,C 180,E1 -17294.68,E2 -17294.68} C_VEL
LIN {X 0,Y 277.348,Z 252.42,A -85,B 0,C 180,E1 -17299.24,E2 -17299.24} C_VEL
LIN {X 0,Y 277.299,Z 252.438,A -85,B 0,C 180,E1 -17304.162,E2 -17304.162} C_VEL
LIN {X 0,Y 277.326,Z 252.435,A -85,B 0,C 180,E1 -17307.507,E2 -17307.507} C_VEL
LIN {X 0,Y 277.257,Z 252.428,A -85,B 0,C 180,E1 -17310.477,E2 -17310.477} C_VEL
LIN {X 0,Y 277.256,Z 252.451,A -85,B 0,C 180,E1 -17313.901,E2 -17313.901} C_VEL
LIN {X 0,Y 277.266,Z 252.434,A -85,B 0,C 180,E1 -17317.476,E2 -17317.476} C_VEL
LIN {X 0,Y 277.221,Z 252.45,A -85,B 0,C 180,E1 -17321.241,E2 -17321.241} C_VEL
LIN {X 0,Y 277.207,Z 252.411,A -85,B 0,C 180,E1 -17325.232,E2 -17325.232} C_VEL
LIN {X 0,Y 277.192,Z 252.459,A -85,B 0,C 180,E1 -17329.527,E2 -17329.527} C_VEL
LIN {X 0,Y 277.246,Z 252.438,A -85,B 0,C 180,E1 -17332.528,E2 -17332.528} C_VEL
LIN {X 0,Y 277.26,Z 252.441,A -85,B 0,C 180,E1 -17336.107,E2 -17336.107} C_VEL
LIN {X 0,Y 277.332,Z 252.663,A -85,B 0,C 180,E1 -17338.354,E2 -17338.354} C_VEL
LIN {X 0,Y 279.358,Z 262.161,A -85,B 0,C 180,E1 -17341.714,E2 -17341.714} C_VEL
LIN {X 0,Y 280.349,Z 267.567,A -85,B 0,C 180,E1 -17343.455,E2 -17343.455} C_VEL
LIN {X 0,Y 283.019,Z 276.324,A -85,B 0,C 180,E1 -17343.955,E2 -17343.955} C_VEL
LIN {X 0,Y 287.658,Z 308.438,A -85,B 0,C 180,E1 -17345.155,E2 -17345.155} C_VEL
LIN {X 0,Y 286.023,Z 375.265,A -85,B 0,C 180,E1 -17346.85,E2 -17346.85} C_VEL
LIN {X 0,Y 285.227,Z 388.532,A -85,B 0,C 180,E1 -17347.452,E2 -17347.452} C_VEL
LIN {X 0,Y 284.159,Z 401.306,A -85,B 0,C 180,E1 -17348.319,E2 -17348.319} C_VEL
LIN {X 0,Y 282.847,Z 413.445,A -85,B 0,C 180,E1 -17349.454,E2 -17349.454} C_VEL
LIN {X 0,Y 281.298,Z 425.004,A -85,B 0,C 180,E1 -17350.858,E2 -17350.858} C_VEL
LIN {X 0,Y 280.047,Z 435.451,A -85,B 0,C 180,E1 -17352.474,E2 -17352.474} C_VEL
LIN {X 0,Y 278.782,Z 444.789,A -85,B 0,C 180,E1 -17354.277,E2 -17354.277} C_VEL
LIN {X 0,Y 277.497,Z 453.839,A -85,B 0,C 180,E1 -17356.452,E2 -17356.452} C_VEL
LIN {X 0,Y 276.526,Z 461.107,A -85,B 0,C 180,E1 -17358.641,E2 -17358.641} C_VEL
LIN {X 0,Y 275.952,Z 465.997,A -85,B 0,C 180,E1 -17360.472,E2 -17360.472} C_VEL
LIN {X 0,Y 275.51,Z 470.735,A -85,B 0,C 180,E1 -17362.673,E2 -17362.673} C_VEL
LIN {X 0,Y 275.243,Z 474.228,A -85,B 0,C 180,E1 -17364.801,E2 -17364.801} C_VEL
LIN {X 0,Y 275.223,Z 476.909,A -85,B 0,C 180,E1 -17367.073,E2 -17367.073} C_VEL
LIN {X 0,Y 275.233,Z 478.114,A -85,B 0,C 180,E1 -17368.537,E2 -17368.537} C_VEL
LIN {X 0,Y 275.23,Z 478.875,A -85,B 0,C 180,E1 -17370,E2 -17370} C_VEL
LIN {X 0,Y 275.233,Z 479.235,A -85,B 0,C 180,E1 -17371.464,E2 -17371.464} C_VEL
LIN {X 0,Y 275.229,Z 479.211,A -85,B 0,C 180,E1 -17372.928,E2 -17372.928} C_VEL
LIN {X 0,Y 275.356,Z 478.249,A -85,B 0,C 180,E1 -17375.451,E2 -17375.451} C_VEL
LIN {X 0,Y 275.624,Z 476.758,A -85,B 0,C 180,E1 -17377.325,E2 -17377.325} C_VEL
LIN {X 0,Y 276.494,Z 473.096,A -85,B 0,C 180,E1 -17380.25,E2 -17380.25} C_VEL
LIN {X 0,Y 277.505,Z 469.156,A -85,B 0,C 180,E1 -17382.432,E2 -17382.432} C_VEL
LIN {X 0,Y 278.813,Z 464.11,A -85,B 0,C 180,E1 -17384.6,E2 -17384.6} C_VEL
LIN {X 0,Y 280.646,Z 457.777,A -85,B 0,C 180,E1 -17386.738,E2 -17386.738} C_VEL
LIN {X 0,Y 282.701,Z 449.892,A -85,B 0,C 180,E1 -17388.856,E2 -17388.856} C_VEL
LIN {X 0,Y 284.613,Z 441.898,A -85,B 0,C 180,E1 -17390.603,E2 -17390.603} C_VEL
LIN {X 0,Y 286.787,Z 433.214,A -85,B 0,C 180,E1 -17392.135,E2 -17392.135} C_VEL
LIN {X 0,Y 289.04,Z 422.635,A -85,B 0,C 180,E1 -17393.653,E2 -17393.653} C_VEL
LIN {X 0,Y 290.981,Z 412.419,A -85,B 0,C 180,E1 -17394.813,E2 -17394.813} C_VEL
LIN {X 0,Y 292.947,Z 400.247,A -85,B 0,C 180,E1 -17395.87,E2 -17395.87} C_VEL
LIN {X 0,Y 294.536,Z 387.522,A -85,B 0,C 180,E1 -17396.673,E2 -17396.673} C_VEL
LIN {X 0,Y 295.589,Z 374.816,A -85,B 0,C 180,E1 -17397.215,E2 -17397.215} C_VEL
LIN {X 0,Y 297.889,Z 312.671,A -85,B 0,C 180,E1 -17398.763,E2 -17398.763} C_VEL
LIN {X 0,Y 294.697,Z 295.257,A -85,B 0,C 180,E1 -17399.702,E2 -17399.702} C_VEL
LIN {X 0,Y 289.167,Z 282.719,A -85,B 0,C 180,E1 -17400.864,E2 -17400.864} C_VEL
LIN {X 0,Y 282.755,Z 270.387,A -85,B 0,C 180,E1 -17402.228,E2 -17402.228} C_VEL
LIN {X 0,Y 281.017,Z 266.817,A -85,B 0,C 180,E1 -17402.686,E2 -17402.686} C_VEL
LIN {X 0,Y 278.898,Z 258.152,A -85,B 0,C 180,E1 -17406.25,E2 -17406.25} C_VEL
LIN {X 0,Y 277.237,Z 252.467,A -85,B 0,C 180,E1 -17408.975,E2 -17408.975} C_VEL
LIN {X 0,Y 277.207,Z 252.439,A -85,B 0,C 180,E1 -17413.199,E2 -17413.199} C_VEL
LIN {X 0,Y 277.22,Z 252.429,A -85,B 0,C 180,E1 -17417.324,E2 -17417.324} C_VEL
LIN {X 0,Y 277.245,Z 252.448,A -85,B 0,C 180,E1 -17420.668,E2 -17420.668} C_VEL
LIN {X 0,Y 277.292,Z 252.439,A -85,B 0,C 180,E1 -17424.336,E2 -17424.336} C_VEL
LIN {X 0,Y 277.253,Z 252.441,A -85,B 0,C 180,E1 -17427.831,E2 -17427.831} C_VEL
LIN {X 0,Y 277.247,Z 252.442,A -85,B 0,C 180,E1 -17431.202,E2 -17431.202} C_VEL
LIN {X 0,Y 277.244,Z 252.449,A -85,B 0,C 180,E1 -17434.467,E2 -17434.467} C_VEL
LIN {X 0,Y 277.261,Z 252.45,A -85,B 0,C 180,E1 -17437.647,E2 -17437.647} C_VEL
LIN {X 0,Y 277.294,Z 252.434,A -85,B 0,C 180,E1 -17440.757,E2 -17440.757} C_VEL
LIN {X 0,Y 277.418,Z 252.418,A -85,B 0,C 180,E1 -17445.319,E2 -17445.319} C_VEL
LIN {X 0,Y 277.464,Z 252.412,A -85,B 0,C 180,E1 -17449.781,E2 -17449.781} C_VEL
LIN {X 0,Y 277.616,Z 252.399,A -85,B 0,C 180,E1 -17452.722,E2 -17452.722} C_VEL
LIN {X 0,Y 277.816,Z 252.367,A -85,B 0,C 180,E1 -17458.544,E2 -17458.544} C_VEL
LIN {X 0,Y 277.816,Z 252.379,A -85,B 0,C 180,E1 -17461.443,E2 -17461.443} C_VEL
LIN {X 0,Y 277.603,Z 252.393,A -85,B 0,C 180,E1 -17467.265,E2 -17467.265} C_VEL
LIN {X 0,Y 277.455,Z 252.421,A -85,B 0,C 180,E1 -17470.206,E2 -17470.206} C_VEL
LIN {X 0,Y 277.402,Z 252.424,A -85,B 0,C 180,E1 -17474.668,E2 -17474.668} C_VEL
LIN {X 0,Y 277.324,Z 252.435,A -85,B 0,C 180,E1 -17479.227,E2 -17479.227} C_VEL
LIN {X 0,Y 277.305,Z 252.439,A -85,B 0,C 180,E1 -17484.163,E2 -17484.163} C_VEL
LIN {X 0,Y 277.304,Z 252.426,A -85,B 0,C 180,E1 -17487.496,E2 -17487.496} C_VEL
LIN {X 0,Y 277.254,Z 252.433,A -85,B 0,C 180,E1 -17490.474,E2 -17490.474} C_VEL
LIN {X 0,Y 277.311,Z 252.463,A -85,B 0,C 180,E1 -17495.338,E2 -17495.338} C_VEL
LIN {X 0,Y 277.439,Z 253.282,A -85,B 0,C 180,E1 -17495.844,E2 -17495.844} C_VEL
LIN {X 0,Y 279.6,Z 260.911,A -85,B 0,C 180,E1 -17499.153,E2 -17499.153} C_VEL
LIN {X 0,Y 286.947,Z 274.347,A -85,B 0,C 180,E1 -17500.781,E2 -17500.781} C_VEL
LIN {X 0,Y 293.553,Z 287.94,A -85,B 0,C 180,E1 -17502.158,E2 -17502.158} C_VEL
LIN {X 0,Y 297.554,Z 297.485,A -85,B 0,C 180,E1 -17502.983,E2 -17502.983} C_VEL
LIN {X 0,Y 298.279,Z 302.215,A -85,B 0,C 180,E1 -17503.217,E2 -17503.217} C_VEL
LIN {X 0,Y 295.706,Z 368.828,A -85,B 0,C 180,E1 -17504.877,E2 -17504.877} C_VEL
LIN {X 0,Y 294.535,Z 382.319,A -85,B 0,C 180,E1 -17505.479,E2 -17505.479} C_VEL
LIN {X 0,Y 293.1,Z 394.575,A -85,B 0,C 180,E1 -17506.301,E2 -17506.301} C_VEL
LIN {X 0,Y 291.37,Z 405.528,A -85,B 0,C 180,E1 -17507.282,E2 -17507.282} C_VEL
LIN {X 0,Y 289.317,Z 416.492,A -85,B 0,C 180,E1 -17508.551,E2 -17508.551} C_VEL
LIN {X 0,Y 286.922,Z 427.747,A -85,B 0,C 180,E1 -17510.214,E2 -17510.214} C_VEL
LIN {X 0,Y 284.731,Z 436.798,A -85,B 0,C 180,E1 -17511.897,E2 -17511.897} C_VEL
LIN {X 0,Y 282.631,Z 445.011,A -85,B 0,C 180,E1 -17513.802,E2 -17513.802} C_VEL
LIN {X 0,Y 280.422,Z 452.887,A -85,B 0,C 180,E1 -17516.086,E2 -17516.086} C_VEL
LIN {X 0,Y 278.91,Z 458.248,A -85,B 0,C 180,E1 -17518.051,E2 -17518.051} C_VEL
LIN {X 0,Y 277.463,Z 463.299,A -85,B 0,C 180,E1 -17520.401,E2 -17520.401} C_VEL
LIN {X 0,Y 276.413,Z 467.176,A -85,B 0,C 180,E1 -17522.841,E2 -17522.841} C_VEL
LIN {X 0,Y 275.899,Z 468.913,A -85,B 0,C 180,E1 -17524.339,E2 -17524.339} C_VEL
LIN {X 0,Y 275.385,Z 470.807,A -85,B 0,C 180,E1 -17526.72,E2 -17526.72} C_VEL
LIN {X 0,Y 275.022,Z 471.647,A -85,B 0,C 180,E1 -17529.037,E2 -17529.037} C_VEL
LIN {X 0,Y 274.92,Z 471.597,A -85,B 0,C 180,E1 -17531.032,E2 -17531.032} C_VEL
LIN {X 0,Y 274.894,Z 470.37,A -85,B 0,C 180,E1 -17533.666,E2 -17533.666} C_VEL
LIN {X 0,Y 275.107,Z 468.105,A -85,B 0,C 180,E1 -17536.073,E2 -17536.073} C_VEL
LIN {X 0,Y 275.461,Z 465.107,A -85,B 0,C 180,E1 -17538.222,E2 -17538.222} C_VEL
LIN {X 0,Y 275.86,Z 460.877,A -85,B 0,C 180,E1 -17540.468,E2 -17540.468} C_VEL
LIN {X 0,Y 276.661,Z 454.399,A -85,B 0,C 180,E1 -17543.069,E2 -17543.069} C_VEL
LIN {X 0,Y 277.618,Z 447.34,A -85,B 0,C 180,E1 -17545.28,E2 -17545.28} C_VEL
LIN {X 0,Y 278.792,Z 438.484,A -85,B 0,C 180,E1 -17547.471,E2 -17547.471} C_VEL
LIN {X 0,Y 280.258,Z 428.388,A -85,B 0,C 180,E1 -17549.461,E2 -17549.461} C_VEL
LIN {X 0,Y 281.602,Z 418.755,A -85,B 0,C 180,E1 -17550.976,E2 -17550.976} C_VEL
LIN {X 0,Y 282.823,Z 408.211,A -85,B 0,C 180,E1 -17552.314,E2 -17552.314} C_VEL
LIN {X 0,Y 284.13,Z 395.709,A -85,B 0,C 180,E1 -17553.545,E2 -17553.545} C_VEL
LIN {X 0,Y 285.061,Z 383.849,A -85,B 0,C 180,E1 -17554.418,E2 -17554.418} C_VEL
LIN {X 0,Y 285.925,Z 370.766,A -85,B 0,C 180,E1 -17555.067,E2 -17555.067} C_VEL
LIN {X 0,Y 286.453,Z 352.755,A -85,B 0,C 180,E1 -17555.587,E2 -17555.587} C_VEL
LIN {X 0,Y 287.886,Z 296.298,A -85,B 0,C 180,E1 -17556.988,E2 -17556.988} C_VEL
LIN {X 0,Y 284.631,Z 277.017,A -85,B 0,C 180,E1 -17557.749,E2 -17557.749} C_VEL
LIN {X 0,Y 279.208,Z 260.749,A -85,B 0,C 180,E1 -17558.638,E2 -17558.638} C_VEL
LIN {X 0,Y 278.251,Z 256.127,A -85,B 0,C 180,E1 -17560.183,E2 -17560.183} C_VEL
LIN {X 0,Y 277.469,Z 252.494,A -85,B 0,C 180,E1 -17561.598,E2 -17561.598} C_VEL
LIN {X 0,Y 277.403,Z 252.43,A -85,B 0,C 180,E1 -17565.725,E2 -17565.725} C_VEL
LIN {X 0,Y 277.337,Z 252.419,A -85,B 0,C 180,E1 -17570.371,E2 -17570.371} C_VEL
LIN {X 0,Y 277.324,Z 252.429,A -85,B 0,C 180,E1 -17574.194,E2 -17574.194} C_VEL
LIN {X 0,Y 277.299,Z 252.402,A -85,B 0,C 180,E1 -17577.514,E2 -17577.514} C_VEL
LIN {X 0,Y 277.279,Z 252.442,A -85,B 0,C 180,E1 -17580.501,E2 -17580.501} C_VEL
LIN {X 0,Y 277.259,Z 252.441,A -85,B 0,C 180,E1 -17583.893,E2 -17583.893} C_VEL
LIN {X 0,Y 277.291,Z 252.441,A -85,B 0,C 180,E1 -17587.465,E2 -17587.465} C_VEL
LIN {X 0,Y 277.273,Z 252.431,A -85,B 0,C 180,E1 -17591.224,E2 -17591.224} C_VEL
LIN {X 0,Y 277.261,Z 252.443,A -85,B 0,C 180,E1 -17595.213,E2 -17595.213} C_VEL
LIN {X 0,Y 277.268,Z 252.431,A -85,B 0,C 180,E1 -17599.5,E2 -17599.5} C_VEL
LIN {X 0,Y 277.264,Z 252.422,A -85,B 0,C 180,E1 -17602.54,E2 -17602.54} C_VEL
LIN {X 0,Y 277.23,Z 252.451,A -85,B 0,C 180,E1 -17606.112,E2 -17606.112} C_VEL
LIN {X 0,Y 277.24,Z 252.439,A -85,B 0,C 180,E1 -17609.545,E2 -17609.545} C_VEL
LIN {X 0,Y 277.294,Z 252.409,A -85,B 0,C 180,E1 -17613.553,E2 -17613.553} C_VEL
LIN {X 0,Y 277.278,Z 252.444,A -85,B 0,C 180,E1 -17617.662,E2 -17617.662} C_VEL
LIN {X 0,Y 277.349,Z 252.431,A -85,B 0,C 180,E1 -17619.861,E2 -17619.861} C_VEL
LIN {X 0,Y 276.662,Z 252.511,A -85,B 0,C 180,E1 -17621.074,E2 -17621.074} C_VEL
LIN {X 0,Y 273.81,Z 252.844,A -85,B 0,C 180,E1 -17623.051,E2 -17623.051} C_VEL
LIN {X 0,Y 271.417,Z 253.132,A -85,B 0,C 180,E1 -17624.658,E2 -17624.658} C_VEL
LIN {X 0,Y 270.413,Z 253.261,A -85,B 0,C 180,E1 -17625.903,E2 -17625.903} C_VEL
LIN {X 0,Y 270.343,Z 253.275,A -85,B 0,C 180,E1 -17626.325,E2 -17626.325} C_VEL
LIN {X 0,Y 270.569,Z 253.281,A -85,B 0,C 180,E1 -17631.041,E2 -17631.041} C_VEL
LIN {X 0,Y 270.537,Z 253.273,A -85,B 0,C 180,E1 -17634.043,E2 -17634.043} C_VEL
LIN {X 0,Y 270.782,Z 253.212,A -85,B 0,C 180,E1 -17638.52,E2 -17638.52} C_VEL
LIN {X 0,Y 270.784,Z 253.242,A -85,B 0,C 180,E1 -17641.494,E2 -17641.494} C_VEL
LIN {X 0,Y 270.567,Z 253.266,A -85,B 0,C 180,E1 -17647.469,E2 -17647.469} C_VEL
LIN {X 0,Y 270.412,Z 253.263,A -85,B 0,C 180,E1 -17650.488,E2 -17650.488} C_VEL
LIN {X 0,Y 270.407,Z 253.3,A -85,B 0,C 180,E1 -17655.071,E2 -17655.071} C_VEL
LIN {X 0,Y 270.306,Z 253.291,A -85,B 0,C 180,E1 -17659.761,E2 -17659.761} C_VEL
LIN {X 0,Y 270.245,Z 253.32,A -85,B 0,C 180,E1 -17664.595,E2 -17664.595} C_VEL
LIN {X 0,Y 270.254,Z 253.315,A -85,B 0,C 180,E1 -17667.917,E2 -17667.917} C_VEL
LIN {X 0,Y 270.184,Z 253.318,A -85,B 0,C 180,E1 -17671.354,E2 -17671.354} C_VEL
LIN {X 0,Y 270.208,Z 253.327,A -85,B 0,C 180,E1 -17674.911,E2 -17674.911} C_VEL
LIN {X 0,Y 270.21,Z 253.32,A -85,B 0,C 180,E1 -17678.715,E2 -17678.715} C_VEL
LIN {X 0,Y 270.184,Z 253.312,A -85,B 0,C 180,E1 -17682.563,E2 -17682.563} C_VEL
LIN {X 0,Y 270.16,Z 253.301,A -85,B 0,C 180,E1 -17686.759,E2 -17686.759} C_VEL
LIN {X 0,Y 270.182,Z 253.318,A -85,B 0,C 180,E1 -17691.301,E2 -17691.301} C_VEL
LIN {X 0,Y 270.212,Z 253.321,A -85,B 0,C 180,E1 -17695.097,E2 -17695.097} C_VEL
LIN {X 0,Y 270.283,Z 253.461,A -85,B 0,C 180,E1 -17697.899,E2 -17697.899} C_VEL
LIN {X 0,Y 272.548,Z 264.364,A -85,B 0,C 180,E1 -17701.875,E2 -17701.875} C_VEL
LIN {X 0,Y 273.127,Z 267.467,A -85,B 0,C 180,E1 -17702.863,E2 -17702.863} C_VEL
LIN {X 0,Y 276.109,Z 276.459,A -85,B 0,C 180,E1 -17703.416,E2 -17703.416} C_VEL
LIN {X 0,Y 278.61,Z 292.183,A -85,B 0,C 180,E1 -17704.049,E2 -17704.049} C_VEL
LIN {X 0,Y 281.015,Z 310.957,A -85,B 0,C 180,E1 -17704.743,E2 -17704.743} C_VEL
LIN {X 0,Y 279.298,Z 375.35,A -85,B 0,C 180,E1 -17706.407,E2 -17706.407} C_VEL
LIN {X 0,Y 278.461,Z 388.55,A -85,B 0,C 180,E1 -17707.021,E2 -17707.021} C_VEL
LIN {X 0,Y 277.439,Z 400.732,A -85,B 0,C 180,E1 -17707.864,E2 -17707.864} C_VEL
LIN {X 0,Y 276.117,Z 412.194,A -85,B 0,C 180,E1 -17708.93,E2 -17708.93} C_VEL
LIN {X 0,Y 274.604,Z 423.985,A -85,B 0,C 180,E1 -17710.373,E2 -17710.373} C_VEL
LIN {X 0,Y 273.251,Z 434.589,A -85,B 0,C 180,E1 -17712.023,E2 -17712.023} C_VEL
LIN {X 0,Y 271.934,Z 444.108,A -85,B 0,C 180,E1 -17713.87,E2 -17713.87} C_VEL
LIN {X 0,Y 270.562,Z 453.254,A -85,B 0,C 180,E1 -17716.098,E2 -17716.098} C_VEL
LIN {X 0,Y 269.528,Z 460.61,A -85,B 0,C 180,E1 -17718.342,E2 -17718.342} C_VEL
LIN {X 0,Y 268.937,Z 465.576,A -85,B 0,C 180,E1 -17720.221,E2 -17720.221} C_VEL
LIN {X 0,Y 268.433,Z 470.381,A -85,B 0,C 180,E1 -17722.478,E2 -17722.478} C_VEL
LIN {X 0,Y 268.149,Z 474.262,A -85,B 0,C 180,E1 -17724.889,E2 -17724.889} C_VEL
LIN {X 0,Y 268.137,Z 476.682,A -85,B 0,C 180,E1 -17726.996,E2 -17726.996} C_VEL
LIN {X 0,Y 268.139,Z 477.917,A -85,B 0,C 180,E1 -17728.499,E2 -17728.499} C_VEL
LIN {X 0,Y 268.157,Z 478.734,A -85,B 0,C 180,E1 -17730,E2 -17730} C_VEL
LIN {X 0,Y 268.139,Z 479.122,A -85,B 0,C 180,E1 -17731.502,E2 -17731.502} C_VEL
LIN {X 0,Y 268.176,Z 478.75,A -85,B 0,C 180,E1 -17734.51,E2 -17734.51} C_VEL
LIN {X 0,Y 268.323,Z 477.985,A -85,B 0,C 180,E1 -17736.014,E2 -17736.014} C_VEL
LIN {X 0,Y 268.943,Z 475.19,A -85,B 0,C 180,E1 -17739.021,E2 -17739.021} C_VEL
LIN {X 0,Y 269.791,Z 471.999,A -85,B 0,C 180,E1 -17741.267,E2 -17741.267} C_VEL
LIN {X 0,Y 270.97,Z 467.771,A -85,B 0,C 180,E1 -17743.499,E2 -17743.499} C_VEL
LIN {X 0,Y 272.886,Z 461.389,A -85,B 0,C 180,E1 -17746.073,E2 -17746.073} C_VEL
LIN {X 0,Y 274.95,Z 454.44,A -85,B 0,C 180,E1 -17748.248,E2 -17748.248} C_VEL
LIN {X 0,Y 277.192,Z 445.611,A -85,B 0,C 180,E1 -17750.446,E2 -17750.446} C_VEL
LIN {X 0,Y 279.403,Z 436.945,A -85,B 0,C 180,E1 -17752.167,E2 -17752.167} C_VEL
LIN {X 0,Y 282.075,Z 426.046,A -85,B 0,C 180,E1 -17753.884,E2 -17753.884} C_VEL
LIN {X 0,Y 284.341,Z 415.053,A -85,B 0,C 180,E1 -17755.237,E2 -17755.237} C_VEL
LIN {X 0,Y 286.511,Z 402.762,A -85,B 0,C 180,E1 -17756.398,E2 -17756.398} C_VEL
LIN {X 0,Y 288.126,Z 391.115,A -85,B 0,C 180,E1 -17757.217,E2 -17757.217} C_VEL
LIN {X 0,Y 289.392,Z 378.047,A -85,B 0,C 180,E1 -17757.848,E2 -17757.848} C_VEL
LIN {X 0,Y 290.253,Z 359.256,A -85,B 0,C 180,E1 -17758.385,E2 -17758.385} C_VEL
LIN {X 0,Y 291.922,Z 313.053,A -85,B 0,C 180,E1 -17759.546,E2 -17759.546} C_VEL
LIN {X 0,Y 288.87,Z 297.223,A -85,B 0,C 180,E1 -17760.457,E2 -17760.457} C_VEL
LIN {X 0,Y 282.62,Z 283.524,A -85,B 0,C 180,E1 -17761.824,E2 -17761.824} C_VEL
LIN {X 0,Y 275.635,Z 270.396,A -85,B 0,C 180,E1 -17763.385,E2 -17763.385} C_VEL
LIN {X 0,Y 273.787,Z 266.625,A -85,B 0,C 180,E1 -17763.91,E2 -17763.91} C_VEL
LIN {X 0,Y 272.085,Z 259.921,A -85,B 0,C 180,E1 -17766.792,E2 -17766.792} C_VEL
LIN {X 0,Y 270.167,Z 253.356,A -85,B 0,C 180,E1 -17770.048,E2 -17770.048} C_VEL
LIN {X 0,Y 270.164,Z 253.316,A -85,B 0,C 180,E1 -17773.242,E2 -17773.242} C_VEL
LIN {X 0,Y 270.178,Z 253.306,A -85,B 0,C 180,E1 -17777.436,E2 -17777.436} C_VEL
LIN {X 0,Y 270.223,Z 253.319,A -85,B 0,C 180,E1 -17781.37,E2 -17781.37} C_VEL
LIN {X 0,Y 270.212,Z 253.321,A -85,B 0,C 180,E1 -17785.09,E2 -17785.09} C_VEL
LIN {X 0,Y 270.198,Z 253.325,A -85,B 0,C 180,E1 -17789.132,E2 -17789.132} C_VEL
LIN {X 0,Y 270.204,Z 253.318,A -85,B 0,C 180,E1 -17792.171,E2 -17792.171} C_VEL
LIN {X 0,Y 270.193,Z 253.318,A -85,B 0,C 180,E1 -17795.559,E2 -17795.559} C_VEL
LIN {X 0,Y 270.234,Z 253.311,A -85,B 0,C 180,E1 -17800.233,E2 -17800.233} C_VEL
LIN {X 0,Y 270.377,Z 253.292,A -85,B 0,C 180,E1 -17804.928,E2 -17804.928} C_VEL
LIN {X 0,Y 270.417,Z 253.288,A -85,B 0,C 180,E1 -17809.512,E2 -17809.512} C_VEL
LIN {X 0,Y 270.576,Z 253.277,A -85,B 0,C 180,E1 -17812.531,E2 -17812.531} C_VEL
LIN {X 0,Y 270.78,Z 253.243,A -85,B 0,C 180,E1 -17818.506,E2 -17818.506} C_VEL
LIN {X 0,Y 270.782,Z 253.255,A -85,B 0,C 180,E1 -17821.48,E2 -17821.48} C_VEL
LIN {X 0,Y 270.564,Z 253.27,A -85,B 0,C 180,E1 -17827.455,E2 -17827.455} C_VEL
LIN {X 0,Y 270.407,Z 253.295,A -85,B 0,C 180,E1 -17830.475,E2 -17830.475} C_VEL
LIN {X 0,Y 270.37,Z 253.298,A -85,B 0,C 180,E1 -17835.059,E2 -17835.059} C_VEL
LIN {X 0,Y 270.286,Z 253.315,A -85,B 0,C 180,E1 -17839.749,E2 -17839.749} C_VEL
LIN {X 0,Y 270.26,Z 253.309,A -85,B 0,C 180,E1 -17844.578,E2 -17844.578} C_VEL
LIN {X 0,Y 270.255,Z 253.309,A -85,B 0,C 180,E1 -17847.902,E2 -17847.902} C_VEL
LIN {X 0,Y 270.165,Z 253.314,A -85,B 0,C 180,E1 -17851.341,E2 -17851.341} C_VEL
LIN {X 0,Y 270.217,Z 253.391,A -85,B 0,C 180,E1 -17854.325,E2 -17854.325} C_VEL
LIN {X 0,Y 272.084,Z 260.123,A -85,B 0,C 180,E1 -17857.596,E2 -17857.596} C_VEL
LIN {X 0,Y 272.562,Z 261.508,A -85,B 0,C 180,E1 -17857.986,E2 -17857.986} C_VEL
LIN {X 0,Y 279.903,Z 274.332,A -85,B 0,C 180,E1 -17859.684,E2 -17859.684} C_VEL
LIN {X 0,Y 287.367,Z 289.328,A -85,B 0,C 180,E1 -17861.314,E2 -17861.314} C_VEL
LIN {X 0,Y 291.962,Z 300.195,A -85,B 0,C 180,E1 -17862.308,E2 -17862.308} C_VEL
LIN {X 0,Y 292.404,Z 303.091,A -85,B 0,C 180,E1 -17862.456,E2 -17862.456} C_VEL
LIN {X 0,Y 289.748,Z 368.962,A -85,B 0,C 180,E1 -17864.125,E2 -17864.125} C_VEL
LIN {X 0,Y 288.51,Z 382.62,A -85,B 0,C 180,E1 -17864.746,E2 -17864.746} C_VEL
LIN {X 0,Y 286.953,Z 395.18,A -85,B 0,C 180,E1 -17865.609,E2 -17865.609} C_VEL
LIN {X 0,Y 284.834,Z 407.704,A -85,B 0,C 180,E1 -17866.787,E2 -17866.787} C_VEL
LIN {X 0,Y 282.765,Z 418.231,A -85,B 0,C 180,E1 -17868.078,E2 -17868.078} C_VEL
LIN {X 0,Y 280.544,Z 428.106,A -85,B 0,C 180,E1 -17869.593,E2 -17869.593} C_VEL
LIN {X 0,Y 278.167,Z 437.324,A -85,B 0,C 180,E1 -17871.356,E2 -17871.356} C_VEL
LIN {X 0,Y 276.033,Z 445.268,A -85,B 0,C 180,E1 -17873.249,E2 -17873.249} C_VEL
LIN {X 0,Y 273.686,Z 453.165,A -85,B 0,C 180,E1 -17875.602,E2 -17875.602} C_VEL
LIN {X 0,Y 271.837,Z 459.396,A -85,B 0,C 180,E1 -17877.995,E2 -17877.995} C_VEL
LIN {X 0,Y 270.347,Z 464.167,A -85,B 0,C 180,E1 -17880.401,E2 -17880.401} C_VEL
LIN {X 0,Y 269.422,Z 467.281,A -85,B 0,C 180,E1 -17882.467,E2 -17882.467} C_VEL
LIN {X 0,Y 268.555,Z 470.112,A -85,B 0,C 180,E1 -17885.246,E2 -17885.246} C_VEL
LIN {X 0,Y 268.269,Z 471.124,A -85,B 0,C 180,E1 -17886.861,E2 -17886.861} C_VEL
LIN {X 0,Y 267.977,Z 471.702,A -85,B 0,C 180,E1 -17888.459,E2 -17888.459} C_VEL
LIN {X 0,Y 267.826,Z 471.705,A -85,B 0,C 180,E1 -17890.823,E2 -17890.823} C_VEL
LIN {X 0,Y 267.771,Z 470.713,A -85,B 0,C 180,E1 -17893.219,E2 -17893.219} C_VEL
LIN {X 0,Y 267.992,Z 468.301,A -85,B 0,C 180,E1 -17895.965,E2 -17895.965} C_VEL
LIN {X 0,Y 268.433,Z 464.503,A -85,B 0,C 180,E1 -17898.675,E2 -17898.675} C_VEL
LIN {X 0,Y 268.873,Z 460.068,A -85,B 0,C 180,E1 -17900.976,E2 -17900.976} C_VEL
LIN {X 0,Y 269.632,Z 454.395,A -85,B 0,C 180,E1 -17903.264,E2 -17903.264} C_VEL
LIN {X 0,Y 270.62,Z 447.308,A -85,B 0,C 180,E1 -17905.531,E2 -17905.531} C_VEL
LIN {X 0,Y 271.834,Z 438.422,A -85,B 0,C 180,E1 -17907.777,E2 -17907.777} C_VEL
LIN {X 0,Y 273.355,Z 428.289,A -85,B 0,C 180,E1 -17909.815,E2 -17909.815} C_VEL
LIN {X 0,Y 274.873,Z 417.885,A -85,B 0,C 180,E1 -17911.465,E2 -17911.465} C_VEL
LIN {X 0,Y 276.245,Z 406.38,A -85,B 0,C 180,E1 -17912.916,E2 -17912.916} C_VEL
LIN {X 0,Y 277.458,Z 394.397,A -85,B 0,C 180,E1 -17914.085,E2 -17914.085} C_VEL
LIN {X 0,Y 278.464,Z 381.832,A -85,B 0,C 180,E1 -17914.977,E2 -17914.977} C_VEL
LIN {X 0,Y 279.267,Z 368.858,A -85,B 0,C 180,E1 -17915.596,E2 -17915.596} C_VEL
LIN {X 0,Y 280.836,Z 313.023,A -85,B 0,C 180,E1 -17917.056,E2 -17917.056} C_VEL
LIN {X 0,Y 281.175,Z 296.873,A -85,B 0,C 180,E1 -17917.472,E2 -17917.472} C_VEL
LIN {X 0,Y 278.2,Z 279.132,A -85,B 0,C 180,E1 -17918.188,E2 -17918.188} C_VEL
LIN {X 0,Y 272.472,Z 262.24,A -85,B 0,C 180,E1 -17919.131,E2 -17919.131} C_VEL
LIN {X 0,Y 271.927,Z 260.478,A -85,B 0,C 180,E1 -17919.297,E2 -17919.297} C_VEL
LIN {X 0,Y 270.458,Z 253.662,A -85,B 0,C 180,E1 -17921.808,E2 -17921.808} C_VEL
LIN {X 0,Y 270.354,Z 253.305,A -85,B 0,C 180,E1 -17922.383,E2 -17922.383} C_VEL
LIN {X 0,Y 270.341,Z 253.31,A -85,B 0,C 180,E1 -17925.905,E2 -17925.905} C_VEL
LIN {X 0,Y 270.284,Z 253.3,A -85,B 0,C 180,E1 -17930.623,E2 -17930.623} C_VEL
LIN {X 0,Y 270.252,Z 253.302,A -85,B 0,C 180,E1 -17934.587,E2 -17934.587} C_VEL
LIN {X 0,Y 270.238,Z 253.283,A -85,B 0,C 180,E1 -17937.912,E2 -17937.912} C_VEL
LIN {X 0,Y 270.227,Z 253.326,A -85,B 0,C 180,E1 -17941.342,E2 -17941.342} C_VEL
LIN {X 0,Y 270.219,Z 253.311,A -85,B 0,C 180,E1 -17944.902,E2 -17944.902} C_VEL
LIN {X 0,Y 270.244,Z 253.321,A -85,B 0,C 180,E1 -17948.737,E2 -17948.737} C_VEL
LIN {X 0,Y 270.237,Z 253.299,A -85,B 0,C 180,E1 -17952.545,E2 -17952.545} C_VEL
LIN {X 0,Y 270.207,Z 253.325,A -85,B 0,C 180,E1 -17956.741,E2 -17956.741} C_VEL
LIN {X 0,Y 270.222,Z 253.309,A -85,B 0,C 180,E1 -17959.454,E2 -17959.454} C_VEL
LIN {X 0,Y 270.232,Z 253.309,A -85,B 0,C 180,E1 -17963.728,E2 -17963.728} C_VEL
LIN {X 0,Y 270.181,Z 253.329,A -85,B 0,C 180,E1 -17966.899,E2 -17966.899} C_VEL
LIN {X 0,Y 270.208,Z 253.301,A -85,B 0,C 180,E1 -17970.393,E2 -17970.393} C_VEL
LIN {X 0,Y 270.245,Z 253.293,A -85,B 0,C 180,E1 -17973.771,E2 -17973.771} C_VEL
LIN {X 0,Y 270.223,Z 253.324,A -85,B 0,C 180,E1 -17977.046,E2 -17977.046} C_VEL
LIN {X 0,Y 270.312,Z 253.31,A -85,B 0,C 180,E1 -17980.253,E2 -17980.253} C_VEL
LIN {X 0,Y 270.385,Z 253.259,A -85,B 0,C 180,E1 -17984.942,E2 -17984.942} C_VEL
LIN {X 0,Y 270.343,Z 253.275,A -85,B 0,C 180,E1 -17986.325,E2 -17986.325} C_VEL
LIN {X 0,Y 269.734,Z 253.368,A -85,B 0,C 180,E1 -17987.571,E2 -17987.571} C_VEL
LIN {X 0,Y 267.006,Z 253.723,A -85,B 0,C 180,E1 -17989.605,E2 -17989.605} C_VEL
LIN {X 0,Y 264.653,Z 254.019,A -85,B 0,C 180,E1 -17991.258,E2 -17991.258} C_VEL
LIN {X 0,Y 263.618,Z 254.144,A -85,B 0,C 180,E1 -17992.536,E2 -17992.536} C_VEL
LIN {X 0,Y 263.52,Z 254.15,A -85,B 0,C 180,E1 -17992.969,E2 -17992.969} C_VEL
LIN {X 0,Y 263.747,Z 254.087,A -85,B 0,C 180,E1 -17998.48,E2 -17998.48} C_VEL
LIN {X 0,Y 263.748,Z 254.118,A -85,B 0,C 180,E1 -18001.534,E2 -18001.534} C_VEL
LIN {X 0,Y 263.53,Z 254.139,A -85,B 0,C 180,E1 -18007.669,E2 -18007.669} C_VEL
LIN {X 0,Y 263.352,Z 254.142,A -85,B 0,C 180,E1 -18010.773,E2 -18010.773} C_VEL
LIN {X 0,Y 263.356,Z 254.178,A -85,B 0,C 180,E1 -18015.484,E2 -18015.484} C_VEL
LIN {X 0,Y 263.269,Z 254.162,A -85,B 0,C 180,E1 -18020.313,E2 -18020.313} C_VEL
LIN {X 0,Y 263.199,Z 254.201,A -85,B 0,C 180,E1 -18025.299,E2 -18025.299} C_VEL
LIN {X 0,Y 263.164,Z 254.186,A -85,B 0,C 180,E1 -18028.738,E2 -18028.738} C_VEL
LIN {X 0,Y 263.138,Z 254.205,A -85,B 0,C 180,E1 -18032.294,E2 -18032.294} C_VEL
LIN {X 0,Y 263.187,Z 254.188,A -85,B 0,C 180,E1 -18036.766,E2 -18036.766} C_VEL
LIN {X 0,Y 263.118,Z 254.21,A -85,B 0,C 180,E1 -18039.877,E2 -18039.877} C_VEL
LIN {X 0,Y 263.116,Z 254.17,A -85,B 0,C 180,E1 -18043.993,E2 -18043.993} C_VEL
LIN {X 0,Y 263.087,Z 254.209,A -85,B 0,C 180,E1 -18048.423,E2 -18048.423} C_VEL
LIN {X 0,Y 263.118,Z 254.196,A -85,B 0,C 180,E1 -18052.097,E2 -18052.097} C_VEL
LIN {X 0,Y 263.167,Z 254.195,A -85,B 0,C 180,E1 -18055.889,E2 -18055.889} C_VEL
LIN {X 0,Y 263.213,Z 254.374,A -85,B 0,C 180,E1 -18057.497,E2 -18057.497} C_VEL
LIN {X 0,Y 265.5,Z 265.173,A -85,B 0,C 180,E1 -18061.545,E2 -18061.545} C_VEL
LIN {X 0,Y 265.92,Z 267.346,A -85,B 0,C 180,E1 -18062.233,E2 -18062.233} C_VEL
LIN {X 0,Y 268.263,Z 274.356,A -85,B 0,C 180,E1 -18062.704,E2 -18062.704} C_VEL
LIN {X 0,Y 270.196,Z 280.687,A -85,B 0,C 180,E1 -18063.049,E2 -18063.049} C_VEL
LIN {X 0,Y 274.354,Z 310.842,A -85,B 0,C 180,E1 -18064.235,E2 -18064.235} C_VEL
LIN {X 0,Y 272.582,Z 375.391,A -85,B 0,C 180,E1 -18065.941,E2 -18065.941} C_VEL
LIN {X 0,Y 271.701,Z 388.54,A -85,B 0,C 180,E1 -18066.566,E2 -18066.566} C_VEL
LIN {X 0,Y 270.609,Z 401.277,A -85,B 0,C 180,E1 -18067.477,E2 -18067.477} C_VEL
LIN {X 0,Y 269.259,Z 412.561,A -85,B 0,C 180,E1 -18068.567,E2 -18068.567} C_VEL
LIN {X 0,Y 267.693,Z 424.262,A -85,B 0,C 180,E1 -18070.044,E2 -18070.044} C_VEL
LIN {X 0,Y 266.27,Z 434.925,A -85,B 0,C 180,E1 -18071.757,E2 -18071.757} C_VEL
LIN {X 0,Y 265.102,Z 443.4,A -85,B 0,C 180,E1 -18073.442,E2 -18073.442} C_VEL
LIN {X 0,Y 263.852,Z 451.293,A -85,B 0,C 180,E1 -18075.343,E2 -18075.343} C_VEL
LIN {X 0,Y 262.634,Z 458.977,A -85,B 0,C 180,E1 -18077.639,E2 -18077.639} C_VEL
LIN {X 0,Y 261.893,Z 465.152,A -85,B 0,C 180,E1 -18079.955,E2 -18079.955} C_VEL
LIN {X 0,Y 261.367,Z 470.027,A -85,B 0,C 180,E1 -18082.274,E2 -18082.274} C_VEL
LIN {X 0,Y 261.072,Z 474.239,A -85,B 0,C 180,E1 -18084.941,E2 -18084.941} C_VEL
LIN {X 0,Y 261.034,Z 476.454,A -85,B 0,C 180,E1 -18086.914,E2 -18086.914} C_VEL
LIN {X 0,Y 261.048,Z 477.719,A -85,B 0,C 180,E1 -18088.458,E2 -18088.458} C_VEL
LIN {X 0,Y 261.085,Z 478.583,A -85,B 0,C 180,E1 -18090.001,E2 -18090.001} C_VEL
LIN {X 0,Y 261.048,Z 479.009,A -85,B 0,C 180,E1 -18091.543,E2 -18091.543} C_VEL
LIN {X 0,Y 261.086,Z 478.694,A -85,B 0,C 180,E1 -18094.632,E2 -18094.632} C_VEL
LIN {X 0,Y 261.254,Z 477.967,A -85,B 0,C 180,E1 -18096.178,E2 -18096.178} C_VEL
LIN {X 0,Y 261.528,Z 476.819,A -85,B 0,C 180,E1 -18097.722,E2 -18097.722} C_VEL
LIN {X 0,Y 262.493,Z 473.284,A -85,B 0,C 180,E1 -18100.803,E2 -18100.803} C_VEL
LIN {X 0,Y 263.646,Z 469.478,A -85,B 0,C 180,E1 -18103.097,E2 -18103.097} C_VEL
LIN {X 0,Y 265.101,Z 464.577,A -85,B 0,C 180,E1 -18105.374,E2 -18105.374} C_VEL
LIN {X 0,Y 267.118,Z 458.426,A -85,B 0,C 180,E1 -18107.613,E2 -18107.613} C_VEL
LIN {X 0,Y 269.343,Z 450.801,A -85,B 0,C 180,E1 -18109.829,E2 -18109.829} C_VEL
LIN {X 0,Y 271.419,Z 443.032,A -85,B 0,C 180,E1 -18111.653,E2 -18111.653} C_VEL
LIN {X 0,Y 274.242,Z 432.498,A -85,B 0,C 180,E1 -18113.605,E2 -18113.605} C_VEL
LIN {X 0,Y 276.84,Z 421.791,A -85,B 0,C 180,E1 -18115.165,E2 -18115.165} C_VEL
LIN {X 0,Y 278.917,Z 411.401,A -85,B 0,C 180,E1 -18116.367,E2 -18116.367} C_VEL
LIN {X 0,Y 281.076,Z 398.932,A -85,B 0,C 180,E1 -18117.453,E2 -18117.453} C_VEL
LIN {X 0,Y 282.81,Z 385.498,A -85,B 0,C 180,E1 -18118.299,E2 -18118.299} C_VEL
LIN {X 0,Y 283.866,Z 371.883,A -85,B 0,C 180,E1 -18118.844,E2 -18118.844} C_VEL
LIN {X 0,Y 286.127,Z 314.322,A -85,B 0,C 180,E1 -18120.323,E2 -18120.323} C_VEL
LIN {X 0,Y 283.472,Z 300.319,A -85,B 0,C 180,E1 -18121.157,E2 -18121.157} C_VEL
LIN {X 0,Y 277.752,Z 287.672,A -85,B 0,C 180,E1 -18122.459,E2 -18122.459} C_VEL
LIN {X 0,Y 270.997,Z 274.782,A -85,B 0,C 180,E1 -18124.043,E2 -18124.043} C_VEL
LIN {X 0,Y 266.613,Z 266.616,A -85,B 0,C 180,E1 -18125.19,E2 -18125.19} C_VEL
LIN {X 0,Y 265.145,Z 261.312,A -85,B 0,C 180,E1 -18127.564,E2 -18127.564} C_VEL
LIN {X 0,Y 263.136,Z 254.241,A -85,B 0,C 180,E1 -18131.2,E2 -18131.2} C_VEL
LIN {X 0,Y 263.099,Z 254.203,A -85,B 0,C 180,E1 -18133.99,E2 -18133.99} C_VEL
LIN {X 0,Y 263.135,Z 254.188,A -85,B 0,C 180,E1 -18138.404,E2 -18138.404} C_VEL
LIN {X 0,Y 263.172,Z 254.199,A -85,B 0,C 180,E1 -18142.099,E2 -18142.099} C_VEL
LIN {X 0,Y 263.166,Z 254.204,A -85,B 0,C 180,E1 -18145.881,E2 -18145.881} C_VEL
LIN {X 0,Y 263.139,Z 254.208,A -85,B 0,C 180,E1 -18149.499,E2 -18149.499} C_VEL
LIN {X 0,Y 263.128,Z 254.205,A -85,B 0,C 180,E1 -18152.989,E2 -18152.989} C_VEL
LIN {X 0,Y 263.127,Z 254.199,A -85,B 0,C 180,E1 -18156.375,E2 -18156.375} C_VEL
LIN {X 0,Y 263.219,Z 254.185,A -85,B 0,C 180,E1 -18159.683,E2 -18159.683} C_VEL
LIN {X 0,Y 263.319,Z 254.171,A -85,B 0,C 180,E1 -18164.514,E2 -18164.514} C_VEL
LIN {X 0,Y 263.356,Z 254.167,A -85,B 0,C 180,E1 -18169.227,E2 -18169.227} C_VEL
LIN {X 0,Y 263.538,Z 254.154,A -85,B 0,C 180,E1 -18172.331,E2 -18172.331} C_VEL
LIN {X 0,Y 263.743,Z 254.119,A -85,B 0,C 180,E1 -18178.466,E2 -18178.466} C_VEL
LIN {X 0,Y 263.747,Z 254.13,A -85,B 0,C 180,E1 -18181.52,E2 -18181.52} C_VEL
LIN {X 0,Y 263.527,Z 254.147,A -85,B 0,C 180,E1 -18187.656,E2 -18187.656} C_VEL
LIN {X 0,Y 263.349,Z 254.172,A -85,B 0,C 180,E1 -18190.759,E2 -18190.759} C_VEL
LIN {X 0,Y 263.316,Z 254.176,A -85,B 0,C 180,E1 -18195.472,E2 -18195.472} C_VEL
LIN {X 0,Y 263.251,Z 254.194,A -85,B 0,C 180,E1 -18200.299,E2 -18200.299} C_VEL
LIN {X 0,Y 263.193,Z 254.179,A -85,B 0,C 180,E1 -18205.284,E2 -18205.284} C_VEL
LIN {X 0,Y 263.162,Z 254.206,A -85,B 0,C 180,E1 -18208.722,E2 -18208.722} C_VEL
LIN {X 0,Y 263.151,Z 254.29,A -85,B 0,C 180,E1 -18213.185,E2 -18213.185} C_VEL
LIN {X 0,Y 264.961,Z 260.491,A -85,B 0,C 180,E1 -18216.356,E2 -18216.356} C_VEL
LIN {X 0,Y 265.462,Z 261.895,A -85,B 0,C 180,E1 -18216.695,E2 -18216.695} C_VEL
LIN {X 0,Y 273.19,Z 275.045,A -85,B 0,C 180,E1 -18218.586,E2 -18218.586} C_VEL
LIN {X 0,Y 279.119,Z 286.498,A -85,B 0,C 180,E1 -18219.958,E2 -18219.958} C_VEL
LIN {X 0,Y 284.943,Z 299.221,A -85,B 0,C 180,E1 -18221.265,E2 -18221.265} C_VEL
LIN {X 0,Y 286.541,Z 303.504,A -85,B 0,C 180,E1 -18221.635,E2 -18221.635} C_VEL
LIN {X 0,Y 283.849,Z 369.123,A -85,B 0,C 180,E1 -18223.341,E2 -18223.341} C_VEL
LIN {X 0,Y 282.572,Z 382.626,A -85,B 0,C 180,E1 -18223.962,E2 -18223.962} C_VEL
LIN {X 0,Y 281.16,Z 394.049,A -85,B 0,C 180,E1 -18224.753,E2 -18224.753} C_VEL
LIN {X 0,Y 278.984,Z 406.494,A -85,B 0,C 180,E1 -18225.9,E2 -18225.9} C_VEL
LIN {X 0,Y 276.692,Z 417.676,A -85,B 0,C 180,E1 -18227.264,E2 -18227.264} C_VEL
LIN {X 0,Y 274.199,Z 428.458,A -85,B 0,C 180,E1 -18228.944,E2 -18228.944} C_VEL
LIN {X 0,Y 271.993,Z 436.592,A -85,B 0,C 180,E1 -18230.512,E2 -18230.512} C_VEL
LIN {X 0,Y 269.443,Z 445.523,A -85,B 0,C 180,E1 -18232.667,E2 -18232.667} C_VEL
LIN {X 0,Y 266.992,Z 453.394,A -85,B 0,C 180,E1 -18235.073,E2 -18235.073} C_VEL
LIN {X 0,Y 265.323,Z 458.643,A -85,B 0,C 180,E1 -18237.111,E2 -18237.111} C_VEL
LIN {X 0,Y 263.669,Z 463.645,A -85,B 0,C 180,E1 -18239.573,E2 -18239.573} C_VEL
LIN {X 0,Y 262.5,Z 467.362,A -85,B 0,C 180,E1 -18242.05,E2 -18242.05} C_VEL
LIN {X 0,Y 261.652,Z 469.943,A -85,B 0,C 180,E1 -18244.547,E2 -18244.547} C_VEL
LIN {X 0,Y 261.297,Z 471.035,A -85,B 0,C 180,E1 -18246.206,E2 -18246.206} C_VEL
LIN {X 0,Y 260.97,Z 471.694,A -85,B 0,C 180,E1 -18247.85,E2 -18247.85} C_VEL
LIN {X 0,Y 260.752,Z 471.811,A -85,B 0,C 180,E1 -18250.593,E2 -18250.593} C_VEL
LIN {X 0,Y 260.66,Z 471.005,A -85,B 0,C 180,E1 -18252.747,E2 -18252.747} C_VEL
LIN {X 0,Y 260.75,Z 469.921,A -85,B 0,C 180,E1 -18254.363,E2 -18254.363} C_VEL
LIN {X 0,Y 261.026,Z 467.428,A -85,B 0,C 180,E1 -18256.77,E2 -18256.77} C_VEL
LIN {X 0,Y 261.396,Z 463.901,A -85,B 0,C 180,E1 -18259.151,E2 -18259.151} C_VEL
LIN {X 0,Y 261.926,Z 459.25,A -85,B 0,C 180,E1 -18261.513,E2 -18261.513} C_VEL
LIN {X 0,Y 262.888,Z 452.177,A -85,B 0,C 180,E1 -18264.246,E2 -18264.246} C_VEL
LIN {X 0,Y 264.011,Z 444.521,A -85,B 0,C 180,E1 -18266.566,E2 -18266.566} C_VEL
LIN {X 0,Y 265.15,Z 436.699,A -85,B 0,C 180,E1 -18268.481,E2 -18268.481} C_VEL
LIN {X 0,Y 266.577,Z 427.438,A -85,B 0,C 180,E1 -18270.319,E2 -18270.319} C_VEL
LIN {X 0,Y 268.2,Z 416.414,A -85,B 0,C 180,E1 -18272.064,E2 -18272.064} C_VEL
LIN {X 0,Y 269.654,Z 404.511,A -85,B 0,C 180,E1 -18273.548,E2 -18273.548} C_VEL
LIN {X 0,Y 270.92,Z 391.759,A -85,B 0,C 180,E1 -18274.743,E2 -18274.743} C_VEL
LIN {X 0,Y 271.93,Z 378.988,A -85,B 0,C 180,E1 -18275.608,E2 -18275.608} C_VEL
LIN {X 0,Y 272.651,Z 365.98,A -85,B 0,C 180,E1 -18276.173,E2 -18276.173} C_VEL
LIN {X 0,Y 274.521,Z 297.894,A -85,B 0,C 180,E1 -18277.955,E2 -18277.955} C_VEL
LIN {X 0,Y 271.754,Z 281.165,A -85,B 0,C 180,E1 -18278.648,E2 -18278.648} C_VEL
LIN {X 0,Y 265.78,Z 263.592,A -85,B 0,C 180,E1 -18279.663,E2 -18279.663} C_VEL
LIN {X 0,Y 264.719,Z 260.529,A -85,B 0,C 180,E1 -18279.943,E2 -18279.943} C_VEL
LIN {X 0,Y 263.321,Z 254.273,A -85,B 0,C 180,E1 -18282.377,E2 -18282.377} C_VEL
LIN {X 0,Y 263.307,Z 254.187,A -85,B 0,C 180,E1 -18286.112,E2 -18286.112} C_VEL
LIN {X 0,Y 263.233,Z 254.181,A -85,B 0,C 180,E1 -18290.886,E2 -18290.886} C_VEL
LIN {X 0,Y 263.179,Z 254.17,A -85,B 0,C 180,E1 -18295.294,E2 -18295.294} C_VEL
LIN {X 0,Y 263.179,Z 254.173,A -85,B 0,C 180,E1 -18298.729,E2 -18298.729} C_VEL
LIN {X 0,Y 263.152,Z 254.207,A -85,B 0,C 180,E1 -18302.285,E2 -18302.285} C_VEL
LIN {X 0,Y 263.181,Z 254.189,A -85,B 0,C 180,E1 -18305.978,E2 -18305.978} C_VEL
LIN {X 0,Y 263.178,Z 254.197,A -85,B 0,C 180,E1 -18309.858,E2 -18309.858} C_VEL
LIN {X 0,Y 263.163,Z 254.189,A -85,B 0,C 180,E1 -18313.975,E2 -18313.975} C_VEL
LIN {X 0,Y 263.186,Z 254.194,A -85,B 0,C 180,E1 -18318.39,E2 -18318.39} C_VEL
LIN {X 0,Y 263.18,Z 254.185,A -85,B 0,C 180,E1 -18323.236,E2 -18323.236} C_VEL
LIN {X 0,Y 263.16,Z 254.203,A -85,B 0,C 180,E1 -18325.897,E2 -18325.897} C_VEL
LIN {X 0,Y 263.129,Z 254.196,A -85,B 0,C 180,E1 -18329.514,E2 -18329.514} C_VEL
LIN {X 0,Y 263.173,Z 254.164,A -85,B 0,C 180,E1 -18333.01,E2 -18333.01} C_VEL
LIN {X 0,Y 263.171,Z 254.195,A -85,B 0,C 180,E1 -18336.394,E2 -18336.394} C_VEL
LIN {X 0,Y 263.273,Z 254.186,A -85,B 0,C 180,E1 -18339.703,E2 -18339.703} C_VEL
LIN {X 0,Y 263.333,Z 254.136,A -85,B 0,C 180,E1 -18344.529,E2 -18344.529} C_VEL
LIN {X 0,Y 263.366,Z 254.171,A -85,B 0,C 180,E1 -18349.242,E2 -18349.242} C_VEL
LIN {X 0,Y 263.566,Z 254.15,A -85,B 0,C 180,E1 -18352.346,E2 -18352.346} C_VEL
LIN {X 0,Y 263.52,Z 254.15,A -85,B 0,C 180,E1 -18352.969,E2 -18352.969} C_VEL
LIN {X 0,Y 262.829,Z 254.232,A -85,B 0,C 180,E1 -18354.244,E2 -18354.244} C_VEL
LIN {X 0,Y 260.034,Z 254.557,A -85,B 0,C 180,E1 -18356.326,E2 -18356.326} C_VEL
LIN {X 0,Y 257.722,Z 254.837,A -85,B 0,C 180,E1 -18358.019,E2 -18358.019} C_VEL
LIN {X 0,Y 256.785,Z 254.962,A -85,B 0,C 180,E1 -18359.329,E2 -18359.329} C_VEL
LIN {X 0,Y 256.736,Z 254.971,A -85,B 0,C 180,E1 -18359.772,E2 -18359.772} C_VEL
LIN {X 0,Y 256.711,Z 254.995,A -85,B 0,C 180,E1 -18361.576,E2 -18361.576} C_VEL
LIN {X 0,Y 256.462,Z 255.03,A -85,B 0,C 180,E1 -18366.3,E2 -18366.3} C_VEL
LIN {X 0,Y 256.429,Z 255.005,A -85,B 0,C 180,E1 -18369.472,E2 -18369.472} C_VEL
LIN {X 0,Y 256.259,Z 255.059,A -85,B 0,C 180,E1 -18374.297,E2 -18374.297} C_VEL
LIN {X 0,Y 256.215,Z 255.065,A -85,B 0,C 180,E1 -18377.568,E2 -18377.568} C_VEL
LIN {X 0,Y 256.16,Z 255.045,A -85,B 0,C 180,E1 -18381.123,E2 -18381.123} C_VEL
LIN {X 0,Y 256.178,Z 255.076,A -85,B 0,C 180,E1 -18385.135,E2 -18385.135} C_VEL
LIN {X 0,Y 256.124,Z 255.065,A -85,B 0,C 180,E1 -18388.59,E2 -18388.59} C_VEL
LIN {X 0,Y 256.084,Z 255.079,A -85,B 0,C 180,E1 -18391.706,E2 -18391.706} C_VEL
LIN {X 0,Y 256.09,Z 255.082,A -85,B 0,C 180,E1 -18395.198,E2 -18395.198} C_VEL
LIN {X 0,Y 256.121,Z 255.067,A -85,B 0,C 180,E1 -18397.274,E2 -18397.274} C_VEL
LIN {X 0,Y 256.067,Z 255.084,A -85,B 0,C 180,E1 -18401.208,E2 -18401.208} C_VEL
LIN {X 0,Y 256.039,Z 255.045,A -85,B 0,C 180,E1 -18405.542,E2 -18405.542} C_VEL
LIN {X 0,Y 256.023,Z 255.092,A -85,B 0,C 180,E1 -18408.791,E2 -18408.791} C_VEL
LIN {X 0,Y 256.114,Z 255.072,A -85,B 0,C 180,E1 -18412.866,E2 -18412.866} C_VEL
LIN {X 0,Y 256.168,Z 255.208,A -85,B 0,C 180,E1 -18417.039,E2 -18417.039} C_VEL
LIN {X 0,Y 258.258,Z 265.086,A -85,B 0,C 180,E1 -18420.861,E2 -18420.861} C_VEL
LIN {X 0,Y 258.698,Z 267.27,A -85,B 0,C 180,E1 -18421.581,E2 -18421.581} C_VEL
LIN {X 0,Y 263.565,Z 281.498,A -85,B 0,C 180,E1 -18422.502,E2 -18422.502} C_VEL
LIN {X 0,Y 267.694,Z 311.668,A -85,B 0,C 180,E1 -18423.728,E2 -18423.728} C_VEL
LIN {X 0,Y 265.891,Z 375.255,A -85,B 0,C 180,E1 -18425.451,E2 -18425.451} C_VEL
LIN {X 0,Y 264.971,Z 388.411,A -85,B 0,C 180,E1 -18426.09,E2 -18426.09} C_VEL
LIN {X 0,Y 263.917,Z 400.591,A -85,B 0,C 180,E1 -18426.976,E2 -18426.976} C_VEL
LIN {X 0,Y 262.396,Z 412.844,A -85,B 0,C 180,E1 -18428.185,E2 -18428.185} C_VEL
LIN {X 0,Y 260.791,Z 424.478,A -85,B 0,C 180,E1 -18429.699,E2 -18429.699} C_VEL
LIN {X 0,Y 259.425,Z 434.514,A -85,B 0,C 180,E1 -18431.353,E2 -18431.353} C_VEL
LIN {X 0,Y 257.957,Z 444.356,A -85,B 0,C 180,E1 -18433.378,E2 -18433.378} C_VEL
LIN {X 0,Y 256.471,Z 453.428,A -85,B 0,C 180,E1 -18435.723,E2 -18435.723} C_VEL
LIN {X 0,Y 255.379,Z 460.721,A -85,B 0,C 180,E1 -18438.089,E2 -18438.089} C_VEL
LIN {X 0,Y 254.654,Z 466.525,A -85,B 0,C 180,E1 -18440.469,E2 -18440.469} C_VEL
LIN {X 0,Y 254.179,Z 471.073,A -85,B 0,C 180,E1 -18442.853,E2 -18442.853} C_VEL
LIN {X 0,Y 253.947,Z 474.514,A -85,B 0,C 180,E1 -18445.238,E2 -18445.238} C_VEL
LIN {X 0,Y 253.935,Z 476.22,A -85,B 0,C 180,E1 -18446.827,E2 -18446.827} C_VEL
LIN {X 0,Y 253.958,Z 477.516,A -85,B 0,C 180,E1 -18448.415,E2 -18448.415} C_VEL
LIN {X 0,Y 253.993,Z 478.414,A -85,B 0,C 180,E1 -18450.001,E2 -18450.001} C_VEL
LIN {X 0,Y 253.958,Z 478.895,A -85,B 0,C 180,E1 -18451.586,E2 -18451.586} C_VEL
LIN {X 0,Y 254.013,Z 478.64,A -85,B 0,C 180,E1 -18454.762,E2 -18454.762} C_VEL
LIN {X 0,Y 254.467,Z 476.855,A -85,B 0,C 180,E1 -18457.938,E2 -18457.938} C_VEL
LIN {X 0,Y 255.506,Z 473.386,A -85,B 0,C 180,E1 -18461.102,E2 -18461.102} C_VEL
LIN {X 0,Y 256.706,Z 469.648,A -85,B 0,C 180,E1 -18463.457,E2 -18463.457} C_VEL
LIN {X 0,Y 258.273,Z 464.818,A -85,B 0,C 180,E1 -18465.791,E2 -18465.791} C_VEL
LIN {X 0,Y 260.383,Z 458.745,A -85,B 0,C 180,E1 -18468.084,E2 -18468.084} C_VEL
LIN {X 0,Y 262.665,Z 451.233,A -85,B 0,C 180,E1 -18470.355,E2 -18470.355} C_VEL
LIN {X 0,Y 264.877,Z 443.588,A -85,B 0,C 180,E1 -18472.216,E2 -18472.216} C_VEL
LIN {X 0,Y 267.572,Z 434.276,A -85,B 0,C 180,E1 -18474.024,E2 -18474.024} C_VEL
LIN {X 0,Y 270.155,Z 423.981,A -85,B 0,C 180,E1 -18475.626,E2 -18475.626} C_VEL
LIN {X 0,Y 272.637,Z 412.582,A -85,B 0,C 180,E1 -18477.023,E2 -18477.023} C_VEL
LIN {X 0,Y 274.847,Z 400.615,A -85,B 0,C 180,E1 -18478.129,E2 -18478.129} C_VEL
LIN {X 0,Y 276.702,Z 387.656,A -85,B 0,C 180,E1 -18478.991,E2 -18478.991} C_VEL
LIN {X 0,Y 277.915,Z 374.64,A -85,B 0,C 180,E1 -18479.579,E2 -18479.579} C_VEL
LIN {X 0,Y 280.342,Z 315.487,A -85,B 0,C 180,E1 -18481.147,E2 -18481.147} C_VEL
LIN {X 0,Y 278.068,Z 303.259,A -85,B 0,C 180,E1 -18481.896,E2 -18481.896} C_VEL
LIN {X 0,Y 272.477,Z 290.874,A -85,B 0,C 180,E1 -18483.232,E2 -18483.232} C_VEL
LIN {X 0,Y 265.987,Z 278.441,A -85,B 0,C 180,E1 -18484.827,E2 -18484.827} C_VEL
LIN {X 0,Y 261.238,Z 270.034,A -85,B 0,C 180,E1 -18486.045,E2 -18486.045} C_VEL
LIN {X 0,Y 259.369,Z 266.344,A -85,B 0,C 180,E1 -18486.647,E2 -18486.647} C_VEL
LIN {X 0,Y 256.752,Z 257.47,A -85,B 0,C 180,E1 -18491.068,E2 -18491.068} C_VEL
LIN {X 0,Y 256.05,Z 255.117,A -85,B 0,C 180,E1 -18492.477,E2 -18492.477} C_VEL
LIN {X 0,Y 256.063,Z 255.066,A -85,B 0,C 180,E1 -18496.666,E2 -18496.666} C_VEL
LIN {X 0,Y 256.086,Z 255.081,A -85,B 0,C 180,E1 -18500.854,E2 -18500.854} C_VEL
LIN {X 0,Y 256.14,Z 255.081,A -85,B 0,C 180,E1 -18502.862,E2 -18502.862} C_VEL
LIN {X 0,Y 256.08,Z 255.086,A -85,B 0,C 180,E1 -18506.702,E2 -18506.702} C_VEL
LIN {X 0,Y 256.066,Z 255.087,A -85,B 0,C 180,E1 -18510.388,E2 -18510.388} C_VEL
LIN {X 0,Y 256.079,Z 255.087,A -85,B 0,C 180,E1 -18513.946,E2 -18513.946} C_VEL
LIN {X 0,Y 256.069,Z 255.087,A -85,B 0,C 180,E1 -18517.397,E2 -18517.397} C_VEL
LIN {X 0,Y 256.139,Z 255.069,A -85,B 0,C 180,E1 -18520.77,E2 -18520.77} C_VEL
LIN {X 0,Y 256.239,Z 255.053,A -85,B 0,C 180,E1 -18524.075,E2 -18524.075} C_VEL
LIN {X 0,Y 256.287,Z 255.06,A -85,B 0,C 180,E1 -18527.321,E2 -18527.321} C_VEL
LIN {X 0,Y 256.441,Z 255.038,A -85,B 0,C 180,E1 -18530.616,E2 -18530.616} C_VEL
LIN {X 0,Y 256.466,Z 255.025,A -85,B 0,C 180,E1 -18533.7,E2 -18533.7} C_VEL
LIN {X 0,Y 256.705,Z 254.995,A -85,B 0,C 180,E1 -18538.424,E2 -18538.424} C_VEL
LIN {X 0,Y 256.71,Z 255.005,A -85,B 0,C 180,E1 -18541.562,E2 -18541.562} C_VEL
LIN {X 0,Y 256.447,Z 255.031,A -85,B 0,C 180,E1 -18546.555,E2 -18546.555} C_VEL
LIN {X 0,Y 256.423,Z 255.044,A -85,B 0,C 180,E1 -18549.458,E2 -18549.458} C_VEL
LIN {X 0,Y 256.231,Z 255.063,A -85,B 0,C 180,E1 -18554.284,E2 -18554.284} C_VEL
LIN {X 0,Y 256.174,Z 255.074,A -85,B 0,C 180,E1 -18557.556,E2 -18557.556} C_VEL
LIN {X 0,Y 256.145,Z 255.075,A -85,B 0,C 180,E1 -18561.112,E2 -18561.112} C_VEL
LIN {X 0,Y 256.174,Z 255.054,A -85,B 0,C 180,E1 -18565.131,E2 -18565.131} C_VEL
LIN {X 0,Y 256.096,Z 255.075,A -85,B 0,C 180,E1 -18569.592,E2 -18569.592} C_VEL
LIN {X 0,Y 256.094,Z 255.182,A -85,B 0,C 180,E1 -18571.938,E2 -18571.938} C_VEL
LIN {X 0,Y 257.813,Z 260.974,A -85,B 0,C 180,E1 -18575.031,E2 -18575.031} C_VEL
LIN {X 0,Y 258.88,Z 263.243,A -85,B 0,C 180,E1 -18575.46,E2 -18575.46} C_VEL
LIN {X 0,Y 261.923,Z 268.094,A -85,B 0,C 180,E1 -18576.253,E2 -18576.253} C_VEL
LIN {X 0,Y 268.507,Z 279.274,A -85,B 0,C 180,E1 -18577.9,E2 -18577.9} C_VEL
LIN {X 0,Y 274.028,Z 290.115,A -85,B 0,C 180,E1 -18579.241,E2 -18579.241} C_VEL
LIN {X 0,Y 279.696,Z 302.57,A -85,B 0,C 180,E1 -18580.572,E2 -18580.572} C_VEL
LIN {X 0,Y 280.837,Z 305.284,A -85,B 0,C 180,E1 -18580.836,E2 -18580.836} C_VEL
LIN {X 0,Y 278.057,Z 368.9,A -85,B 0,C 180,E1 -18582.505,E2 -18582.505} C_VEL
LIN {X 0,Y 276.732,Z 382.455,A -85,B 0,C 180,E1 -18583.131,E2 -18583.131} C_VEL
LIN {X 0,Y 275.104,Z 394.864,A -85,B 0,C 180,E1 -18584.002,E2 -18584.002} C_VEL
LIN {X 0,Y 272.871,Z 407.061,A -85,B 0,C 180,E1 -18585.165,E2 -18585.165} C_VEL
LIN {X 0,Y 270.374,Z 418.635,A -85,B 0,C 180,E1 -18586.62,E2 -18586.62} C_VEL
LIN {X 0,Y 267.861,Z 428.825,A -85,B 0,C 180,E1 -18588.258,E2 -18588.258} C_VEL
LIN {X 0,Y 265.071,Z 438.584,A -85,B 0,C 180,E1 -18590.241,E2 -18590.241} C_VEL
LIN {X 0,Y 262.449,Z 447.238,A -85,B 0,C 180,E1 -18592.467,E2 -18592.467} C_VEL
LIN {X 0,Y 260.238,Z 453.909,A -85,B 0,C 180,E1 -18594.619,E2 -18594.619} C_VEL
LIN {X 0,Y 258.235,Z 459.779,A -85,B 0,C 180,E1 -18597.022,E2 -18597.022} C_VEL
LIN {X 0,Y 256.583,Z 464.51,A -85,B 0,C 180,E1 -18599.553,E2 -18599.553} C_VEL
LIN {X 0,Y 255.363,Z 468.008,A -85,B 0,C 180,E1 -18602.104,E2 -18602.104} C_VEL
LIN {X 0,Y 254.758,Z 469.711,A -85,B 0,C 180,E1 -18603.807,E2 -18603.807} C_VEL
LIN {X 0,Y 254.272,Z 471.079,A -85,B 0,C 180,E1 -18605.775,E2 -18605.775} C_VEL
LIN {X 0,Y 253.761,Z 471.998,A -85,B 0,C 180,E1 -18608.897,E2 -18608.897} C_VEL
LIN {X 0,Y 253.652,Z 471.884,A -85,B 0,C 180,E1 -18610.58,E2 -18610.58} C_VEL
LIN {X 0,Y 253.586,Z 471.292,A -85,B 0,C 180,E1 -18612.25,E2 -18612.25} C_VEL
LIN {X 0,Y 253.608,Z 470.283,A -85,B 0,C 180,E1 -18613.911,E2 -18613.911} C_VEL
LIN {X 0,Y 253.76,Z 468.679,A -85,B 0,C 180,E1 -18615.736,E2 -18615.736} C_VEL
LIN {X 0,Y 254.135,Z 465.83,A -85,B 0,C 180,E1 -18618.029,E2 -18618.029} C_VEL
LIN {X 0,Y 254.547,Z 461.735,A -85,B 0,C 180,E1 -18620.464,E2 -18620.464} C_VEL
LIN {X 0,Y 255.351,Z 455.885,A -85,B 0,C 180,E1 -18623.095,E2 -18623.095} C_VEL
LIN {X 0,Y 256.411,Z 448.503,A -85,B 0,C 180,E1 -18625.677,E2 -18625.677} C_VEL
LIN {X 0,Y 257.709,Z 439.906,A -85,B 0,C 180,E1 -18628.046,E2 -18628.046} C_VEL
LIN {X 0,Y 259.13,Z 431.021,A -85,B 0,C 180,E1 -18629.999,E2 -18629.999} C_VEL
LIN {X 0,Y 260.825,Z 420.063,A -85,B 0,C 180,E1 -18631.93,E2 -18631.93} C_VEL
LIN {X 0,Y 262.297,Z 409.055,A -85,B 0,C 180,E1 -18633.456,E2 -18633.456} C_VEL
LIN {X 0,Y 263.692,Z 396.707,A -85,B 0,C 180,E1 -18634.777,E2 -18634.777} C_VEL
LIN {X 0,Y 264.853,Z 383.697,A -85,B 0,C 180,E1 -18635.806,E2 -18635.806} C_VEL
LIN {X 0,Y 265.786,Z 370.369,A -85,B 0,C 180,E1 -18636.5,E2 -18636.5} C_VEL
LIN {X 0,Y 266.441,Z 350.192,A -85,B 0,C 180,E1 -18637.102,E2 -18637.102} C_VEL
LIN {X 0,Y 267.848,Z 298.514,A -85,B 0,C 180,E1 -18638.474,E2 -18638.474} C_VEL
LIN {X 0,Y 265.318,Z 283.191,A -85,B 0,C 180,E1 -18639.131,E2 -18639.131} C_VEL
LIN {X 0,Y 259.605,Z 266.391,A -85,B 0,C 180,E1 -18640.138,E2 -18640.138} C_VEL
LIN {X 0,Y 257.569,Z 260.966,A -85,B 0,C 180,E1 -18640.549,E2 -18640.549} C_VEL
LIN {X 0,Y 256.562,Z 256.341,A -85,B 0,C 180,E1 -18642.256,E2 -18642.256} C_VEL
LIN {X 0,Y 256.294,Z 255.093,A -85,B 0,C 180,E1 -18642.873,E2 -18642.873} C_VEL
